// TwinCAT 3 PLC project Struckig_unittest
// ProjectVersion: 0.19.4.0
// ProgramVersion: 3.1.4026.18
// libraries:
//   Struckig, 0.12.2.0 (Stefan Besler)
//   Tc2_System, * (Beckhoff Automation GmbH)
//   Tc3_Module, * (Beckhoff Automation GmbH)
//   TcUnit_Zeugwerk, 1.3.2 (Zeugwerk GmbH)
// project tree:
//   / PlcTask.TcTTO (not stored)
//   POUs/ DebuggedExamplesTest.TcPOU, KnownExamplesSecondOrderTest.TcPOU, MaxVelocitySwitchingTest.TcPOU, Otg1Test.TcPOU, RandomTest.TcPOU, SetVector3.TcPOU (not stored), PropagateTest.TcPOU, VelocityInterfaceTest.TcPOU, MinDurationTest.TcPOU, MathTest.TcPOU, TargetPosTest.TcPOU, TargetPosAccTest.TcPOU, TargetPosVelTest.TcPOU, TargetPosVelAccTest.TcPOU, SecondaryFeaturesTest.TcPOU, CheckCalculation.TcPOU, KnownExamplesTest.TcPOU, MAIN.TcPOU, ZeroLimitsTest.TcPOU
//   Randomizer/ Randomizer.TcPOU (not stored)
//   Random/ IRandom.TcIO (not stored), RandomGaussian.TcPOU, RandomUniform.TcPOU
//   Random/_Test/ RandomGaussianTest.TcPOU (not stored)
// real-time tasks:
//   TASK PlcTask: cycle T#10ms, priority 20, ADS port 350

// ---- POUs/DebuggedExamplesTest.TcPOU
FUNCTION_BLOCK DebuggedExamplesTest EXTENDS TcUnit_Zeugwerk.FB_TestSuite

Test_Trajectory_HasTargetVelocity_HasTargetAcceleration();

METHOD Test_Trajectory_HasTargetVelocity_HasTargetAcceleration
VAR_INST
  ruckig : Struckig.Otg(0.001, 3) := (
  
    Synchronization := SynchronizationType.TimeSync,        
    MaxVelocity := [ 2000.00000000000000000000, 2000.00000000000000000000, 2000.00000000000000000000 ],
    MaxAcceleration := [ 20000.00000000000000000000, 20000.00000000000000000000, 20000.00000000000000000000 ],
    MaxJerk := [ 800000.00000000000000000000, 800000.00000000000000000000, 800000.00000000000000000000 ],
    CurrentPosition := [ -54.94342725690739825950, -71.16344937395382430623, -99.92141940871530891854 ],
    CurrentVelocity := [ 203.04708462957614756306, -87.88615914847480325989, -244.40742200449426491105 ],
    CurrentAcceleration := [ -9414.24830241836389177479, 3433.58972946014000626747, -1048.10905719350193976425 ],
    TargetPosition := [ -30.34627507739200780179, 41.33313071646210801191, 94.47974487226861128875 ],
    TargetVelocity := [ -104.33706621689987059654, -659.36109838358197521302, 811.33117925934993763804 ],
    TargetAcceleration := [ 523.43053514200096287823, 100.75104632855459385610, 320.80199262854853259341 ]
  );
  
  positionExtrema : Struckig.ProfileBound;
END_VAR
TEST('Trajectory_Profile[1]_Step2_TimeVel');

ruckig();

// Check total duration of profiles
AssertEquals_LREAL(Expected := 0.22338925049474450679, Actual := ruckig.Duration, DELTA := 1E-8, Message := 'Duration incorrect');

// Check duration for each phase
positionExtrema := ruckig._profiles[0].Bound();
AssertEquals_LREAL(0.20657109030979783904, positionExtrema.Tmax, 1E-9, message:='Profile[0] Tmax incorrect');
AssertEquals_LREAL(-29.15176131633907630203, positionExtrema.Maximum, 1E-9, message:='Profile[0] maximum incorrect');
AssertEquals_LREAL(0.00000000000000000000, positionExtrema.Tmin, 1E-9, message:='Profile[0] Tmin incorrect');
AssertEquals_LREAL(-54.94342725690739825950, positionExtrema.Minimum, 1E-9, message:='Profile[0] minimum incorrect');

positionExtrema := ruckig._profiles[1].Bound();
AssertEquals_LREAL(0.19826331168683380968, positionExtrema.Tmax, 1E-9, message:='Profile[1] Tmax incorrect');
AssertEquals_LREAL(55.81702313192161568622, positionExtrema.Maximum, 1E-9, message:='Profile[1] maximum incorrect');
AssertEquals_LREAL(0.01113968648909354625, positionExtrema.Tmin, 1E-9, message:='Profile[1] Tmin incorrect');
AssertEquals_LREAL(-71.74511835894615785492, positionExtrema.Minimum, 1E-9, message:='Profile[1] minimum incorrect');

positionExtrema := ruckig._profiles[2].Bound();
AssertEquals_LREAL(0.22338925049474447904, positionExtrema.Tmax, 1E-9, message:='Profile[2] Tmax incorrect');
AssertEquals_LREAL(94.47974487226861128875, positionExtrema.Maximum, 1E-9, message:='Profile[2] maximum incorrect');
AssertEquals_LREAL(0.02606362117094545780, positionExtrema.Tmin, 1E-9, message:='Profile[2] Tmin incorrect');
AssertEquals_LREAL(-104.28684661857214166503, positionExtrema.Minimum, 1E-9, message:='Profile[2] minimum incorrect');
   

TEST_FINISHED();
END_METHOD

END_FUNCTION_BLOCK

// ---- POUs/KnownExamplesSecondOrderTest.TcPOU
FUNCTION_BLOCK KnownExamplesSecondOrderTest EXTENDS TcUnit_Zeugwerk.FB_TestSuite

example01();
example02();
example03();
example04();
example05();
example06();

METHOD example01
VAR_INST
  otg : Struckig.Otg(0.004, 3) := (  
    MaxVelocity :=         [ 1.0, 1.0, 1.0 ],
    MaxAcceleration :=     [ 1.0, 1.0, 1.0 ],
    MaxJerk :=             [ Struckig.Constants.Infinity, Struckig.Constants.Infinity, Struckig.Constants.Infinity ],
    CurrentPosition :=     [ 0.0, -2.0, 0.0 ],
    CurrentVelocity :=     [ 0.0, 0.0, 0.0 ],
    CurrentAcceleration := [ 0.0, 0.0, 0.0 ],
    TargetPosition :=      [ 1.0, -3.0, 2.0 ],
    TargetVelocity :=      [ 0.0, 0.0, 0.0 ],
    TargetAcceleration :=  [ 0.0, 0.0, 0.0 ]
  );
  
END_VAR
TEST('Example-01');

otg();
AssertEquals_LREAL(Expected := 3.0,
             Actual := CheckCalculation(otg),
             DELTA := 1E-8,
             Message := '');
 
TEST_FINISHED();
END_METHOD

METHOD example02
VAR_INST
  otg : Struckig.Otg(0.004, 3) := (  
    MaxVelocity :=         [ 10.0, 10.0, 10.0 ],
    MaxAcceleration :=     [ 1.0, 1.0, 1.0 ],
    CurrentPosition :=     [ 0.0, -2.0, 1.0 ],
    CurrentVelocity :=     [ 0.0, 0.0, 0.0 ],
    CurrentAcceleration := [ 0.0, 0.0, 0.0 ],
    TargetPosition :=      [ 1.0, -3.0, 2.0 ],
    TargetVelocity :=      [ 1.0, 0.0, 0.0 ],
    TargetAcceleration :=  [ 0.0, 0.5, 0.0 ]
  );
  
END_VAR
TEST('Example-02');

otg();
AssertEquals_LREAL(Expected := 2.0,
             Actual := CheckCalculation(otg),
             Delta := 1E-8,
             Message := '');
 
TEST_FINISHED();
END_METHOD

METHOD example03
VAR_INST
  otg : Struckig.Otg(0.004, 3) := (  
    MaxVelocity :=         [ 10.0, 10.0, 10.0 ],
    MaxAcceleration :=     [ 1.0, 1.0, 1.0 ],
    CurrentPosition :=     [ 0.0, -2.0, -2.0 ],
    CurrentVelocity :=     [ 0.1, 0.1, 1.0 ],
    CurrentAcceleration := [ 0.0, 0.0, 0.0 ],
    TargetPosition :=      [ 1.0, -3.0, 2.0 ],
    TargetVelocity :=      [ 1.0, 0.0, 0.0 ],
    TargetAcceleration :=  [ 0.0, 0.5, 0.0 ]
  );
  
END_VAR
TEST('Example-03');

otg();
AssertEquals_LREAL(Expected := 3.24264068711928,
             Actual := CheckCalculation(otg),
             DELTA := 1E-8,
             Message := '');
 
TEST_FINISHED();
END_METHOD

METHOD example04
VAR_INST
  otg : Struckig.Otg(0.004, 3) := (       
    MaxVelocity :=         [ 10.0, 10.0, 10.0 ],
    MaxAcceleration :=     [ 1.0, 1.0, 1.0 ],
    CurrentPosition :=     [ 0.0, 0.0, 0.0 ],
    CurrentVelocity :=     [ 0.0, 1.0, 0.0 ],
    CurrentAcceleration := [ 0.0, 0.0, 0.0 ],
    TargetPosition :=      [ 0.0, 0.0, 0.0 ],
    TargetVelocity :=      [ 0.0, 1.0, 0.0 ],
    TargetAcceleration :=  [ 0.0, 0.0, 0.0 ]
  );
  
  
END_VAR
TEST('Example-04');

otg();
AssertEquals_LREAL(Expected := 0.0,
             Actual := CheckCalculation(otg),
             DELTA := 1E-8,
             Message := '');
 
TEST_FINISHED();
END_METHOD

METHOD example05
VAR_INST
  otg : Struckig.Otg(0.004, 3) := (  
    MaxVelocity :=         [ 10.0, 10.0, 10.0 ],
    MaxAcceleration :=     [ 1.0, 1.0, 1.0 ],
    CurrentPosition :=     [ 0.0, 0.0, 0.0 ],
    CurrentVelocity :=     [ 0.0, 1.0, 0.0 ],
    CurrentAcceleration := [ 0.0, 0.0, 0.0 ],
    TargetPosition :=      [ 0.0, 1E-4, 0.0 ],
    TargetVelocity :=      [ 0.0, 1.0, 0.0 ],
    TargetAcceleration :=  [ 0.0, 0.0, 0.0 ]
  );
  
END_VAR
TEST('Example-05');

otg();
AssertEquals_LREAL(Expected := 0.0001,
             Actual := CheckCalculation(otg),
             DELTA := 1E-8,
             Message := '');
 
TEST_FINISHED();
END_METHOD

METHOD example06
VAR_INST
  otg : Struckig.Otg(0.004, 3) := (  
    MaxVelocity :=         [ 10.0, 10.0, 10.0 ],
    MaxAcceleration :=     [ 1.0, 1.0, 1.0 ],
    CurrentPosition :=     [ 0.0, 0.0, 0.0 ],
    CurrentVelocity :=     [ 0.0, 1.0, 0.0 ],
    CurrentAcceleration := [ 0.0, 0.0, 0.0 ],
    TargetPosition :=      [ 1E-4, 0.0, 0.0 ],
    TargetVelocity :=      [ 0.0, 1.0, 0.0 ],
    TargetAcceleration :=  [ 0.0, 0.0, 0.0 ]
  );
  
END_VAR
TEST('Example-06');

otg();
AssertEquals_LREAL(Expected := 4.0,
             Actual := CheckCalculation(otg),
             DELTA := 1E-8,
             Message := '');
 
TEST_FINISHED();
END_METHOD

END_FUNCTION_BLOCK

// ---- POUs/CheckCalculation.TcPOU
FUNCTION CheckCalculation : LREAL
VAR_INPUT
  otg : Struckig.IOtg;
END_VAR

REPEAT 
  otg.Cyclic();
  otg.PassOutputToInput();
UNTIL otg.State <> Struckig.TrajectoryState.Busy END_REPEAT

CheckCalculation := otg.Duration;

END_FUNCTION

// ---- POUs/MaxVelocitySwitchingTest.TcPOU
FUNCTION_BLOCK MaxVelocitySwitchingTest EXTENDS TcUnit_Zeugwerk.FB_TestSuite

Test_Trajectory();
Test_SmoothBrake_DuringAccel();
Test_SmoothBrake_FromCruise();
Test_SmoothBrake_Disabled();
Test_SmoothBrake_ReachesNewVelocity();

METHOD Test_SmoothBrake_Disabled
VAR_INST
  otg : Struckig.Otg(0.001, 1) := (
    Synchronization := SynchronizationType.TimeSync,
    SmoothBrake := FALSE,
    MaxVelocity := [ 1000 ],
    MaxAcceleration := [ 5000 ],
    MaxJerk := [ 50000 ],
    CurrentPosition := [ 0 ],
    CurrentVelocity := [ 0 ],
    CurrentAcceleration := [ 0 ],
    TargetPosition := [ 50000 ],
    TargetVelocity := [ 0 ],
    TargetAcceleration := [ 0 ]
  );
END_VAR
TEST('SmoothBrake_Disabled');

otg();

REPEAT 
  otg.Cyclic();
  otg.PassOutputToInput();
UNTIL otg.CurrentTime >= otg._profiles[0].t_sum[2] + 0.05 END_REPEAT

otg.MaxVelocity[0] := 500;

REPEAT 
  otg.Cyclic();
  otg.PassOutputToInput();
UNTIL otg.State <> Struckig.TrajectoryState.Busy END_REPEAT

AssertTrue(otg.State <> Struckig.TrajectoryState.Error, Message := 'Legacy mode (SmoothBrake=FALSE) must complete without error');

TEST_FINISHED();
END_METHOD

METHOD Test_SmoothBrake_DuringAccel
VAR_INST
  otg : Struckig.Otg(0.001, 1) := (
    Synchronization := SynchronizationType.TimeSync,
    SmoothBrake := TRUE,
    MaxVelocity := [ 1000 ],
    MaxAcceleration := [ 5000 ],
    MaxJerk := [ 50000 ],
    CurrentPosition := [ 0 ],
    CurrentVelocity := [ 0 ],
    CurrentAcceleration := [ 0 ],
    TargetPosition := [ 50000 ],
    TargetVelocity := [ 0 ],
    TargetAcceleration := [ 0 ]
  );
END_VAR
VAR_INST
  minV : LREAL;
END_VAR
TEST('SmoothBrake_DuringAccel');

otg();

REPEAT 
  otg.Cyclic();
  otg.PassOutputToInput();
UNTIL otg.NewVelocity[0] > 900 OR_ELSE otg.CurrentTime > 5.0 END_REPEAT

otg.MaxVelocity[0] := 500;

minV := 1000;
REPEAT 
  otg.Cyclic();
  IF otg.CurrentTime < otg._profiles[0].Brake.Duration + otg._profiles[0].t_sum[3] THEN
    IF otg.NewVelocity[0] < minV THEN
      minV := otg.NewVelocity[0];
    END_IF
  END_IF
  otg.PassOutputToInput();
UNTIL otg.State <> Struckig.TrajectoryState.Busy END_REPEAT

AssertTrue(otg.State <> Struckig.TrajectoryState.Error, Message := 'OTG must not enter Error state');
AssertTrue(minV > 400.0, Message := 'During accel, velocity must not dip far below new MaxVelocity (500)');

TEST_FINISHED();
END_METHOD

METHOD Test_SmoothBrake_FromCruise
VAR_INST
  otg : Struckig.Otg(0.001, 1) := (
    Synchronization := SynchronizationType.TimeSync,
    SmoothBrake := TRUE,
    MaxVelocity := [ 1000 ],
    MaxAcceleration := [ 5000 ],
    MaxJerk := [ 50000 ],
    CurrentPosition := [ 0 ],
    CurrentVelocity := [ 0 ],
    CurrentAcceleration := [ 0 ],
    TargetPosition := [ 50000 ],
    TargetVelocity := [ 0 ],
    TargetAcceleration := [ 0 ]
  );
END_VAR
VAR
  minV : LREAL;
END_VAR
TEST('SmoothBrake_FromCruise');

otg();

REPEAT 
  otg.Cyclic();
  otg.PassOutputToInput();
UNTIL otg.CurrentTime >= otg._profiles[0].t_sum[2] + 0.05 END_REPEAT

otg.MaxVelocity[0] := 500;

minV := 1000;
REPEAT 
  otg.Cyclic();
  IF otg.CurrentTime < otg._profiles[0].Brake.Duration + otg._profiles[0].t_sum[3] THEN
    IF otg.NewVelocity[0] < minV THEN
      minV := otg.NewVelocity[0];
    END_IF
  END_IF
  otg.PassOutputToInput();
UNTIL otg.State <> Struckig.TrajectoryState.Busy END_REPEAT

AssertTrue(otg.State <> Struckig.TrajectoryState.Error, Message := 'OTG must not enter Error state');
AssertTrue(minV > 400.0, Message := 'From cruise, velocity must not dip far below new MaxVelocity (500)');

TEST_FINISHED();
END_METHOD

METHOD Test_SmoothBrake_ReachesNewVelocity
VAR_INST
  otg : Struckig.Otg(0.001, 1) := (
    Synchronization := SynchronizationType.TimeSync,
    SmoothBrake := TRUE,
    MaxVelocity := [ 1000 ],
    MaxAcceleration := [ 5000 ],
    MaxJerk := [ 50000 ],
    CurrentPosition := [ 0 ],
    CurrentVelocity := [ 0 ],
    CurrentAcceleration := [ 0 ],
    TargetPosition := [ 50000 ],
    TargetVelocity := [ 0 ],
    TargetAcceleration := [ 0 ]
  );
END_VAR
VAR
  vAfter : LREAL;
  captured : BOOL;
END_VAR
TEST('SmoothBrake_ReachesNewVelocity');

otg();

REPEAT 
  otg.Cyclic();
  otg.PassOutputToInput();
UNTIL otg.CurrentTime >= otg._profiles[0].t_sum[2] + 0.05 END_REPEAT

otg.MaxVelocity[0] := 500;

captured := FALSE;
REPEAT 
  otg.Cyclic();
  IF NOT captured AND_THEN otg.CurrentTime >= otg._profiles[0].Brake.Duration + otg._profiles[0].t_sum[2] + 0.01 THEN
    vAfter := otg.NewVelocity[0];
    captured := TRUE;
  END_IF
  otg.PassOutputToInput();
UNTIL otg.State <> Struckig.TrajectoryState.Busy END_REPEAT

AssertTrue(otg.State <> Struckig.TrajectoryState.Error, Message := 'OTG must not enter Error state');
AssertTrue(vAfter > 490.0 AND_THEN vAfter < 510.0, Message := 'After transition, velocity should settle at new MaxVelocity (~500)');

TEST_FINISHED();
END_METHOD

METHOD Test_Trajectory
VAR_INST
  ruckig : Struckig.Otg(0.001, 1) := (
    Synchronization := SynchronizationType.TimeSync,        
    MaxVelocity := [ 10000.00000000000000000000 ],
    MaxAcceleration := [ 20000.00000000000000000000 ],
    MaxJerk := [ 800000.00000000000000000000 ],
    CurrentPosition := [ 0 ],
    CurrentVelocity := [ 0 ],
    CurrentAcceleration := [ 0 ],
    TargetPosition := [ 10000 ],
    TargetVelocity := [ 0 ],
    TargetAcceleration := [ 0 ]
  );
  
END_VAR
TEST('Trajectory');

ruckig();

REPEAT 
  ruckig.Cyclic();
  ruckig.PassOutputToInput();
UNTIL ruckig.CurrentTime >= ruckig._profiles[0].t_sum[2] + 0.05 END_REPEAT

ruckig.MaxVelocity[0] := 9500;

REPEAT 
  ruckig.Cyclic();
  ruckig.PassOutputToInput();
UNTIL ruckig.State <> Struckig.TrajectoryState.Busy END_REPEAT

TEST_FINISHED();
END_METHOD

END_FUNCTION_BLOCK

// ---- POUs/Otg1Test.TcPOU
FUNCTION_BLOCK Otg1Test EXTENDS TcUnit_Zeugwerk.FB_TestSuite

example06();

METHOD example06
VAR_INST
  otg1 : Struckig.Otg1(0.005) := (
  
    Synchronization := SynchronizationType.None,        
    MaxVelocity :=          0.4,
    MaxAcceleration :=      1.0,
    MaxJerk :=              2.0,
    CurrentPosition :=      0.0,
    CurrentVelocity :=      0.0,
    CurrentAcceleration :=  0.0,
    TargetPosition :=       1.0,
    TargetVelocity :=       0.0,
    TargetAcceleration :=   0.0
  );
  	
END_VAR
TEST('Example-06');

otg1();
AssertEquals_LREAL(Expected := 3.394427191,
             Actual := CheckCalculation(otg1),
             DELTA := 1E-8,
             Message := '');
 
TEST_FINISHED();
END_METHOD

END_FUNCTION_BLOCK

// ---- POUs/RandomTest.TcPOU
FUNCTION_BLOCK RandomTest EXTENDS TcUnit_Zeugwerk.FB_TestSuite
VAR
  _number_trajectories : UDINT := 256 * 1024; // Some user variable you want to be able to set
  _position_random_3 : UDINT  := MIN(250000, _number_trajectories / 25);  
  _velocity_random_3 : UDINT  := MIN(250000, _number_trajectories / 25);
  
  _positionDist : RandomGaussian(seed:=45, mu:=0, sigma:=4);
  _dynamicDist : RandomGaussian(seed:=46, mu:=0, sigma:=0.8);
  _limitDist : RandomUniform(seed:=47, lowerBound:=0.08, upperBound:=16.0);
  _limitDistHigh : RandomUniform(seed:=48, lowerBound:=10, upperBound:=1000000.0);
  _minLimitDist : RandomUniform(seed:=49, lowerBound:=-16, upperBound:=-0.08);

END_VAR

Test_PositionFirstRandom3();

Test_VelocitySecondRandom3();
Test_PositionSecondRandom3();

Test_VelocityThirdRandom3();
Test_PositionThirdRandom3();

METHOD Test_PositionFirstRandom3
VAR_INST
  p : Randomizer(_positionDist);
  d : Randomizer(_dynamicDist);
  l : Randomizer(_limitDist);
  
  otg : Struckig.Otg(0.005, 3) := (
    ControlInterface := ControlInterfaceType.Position
  );
   
END_VAR
VAR
  i : UDINT;
END_VAR
TEST('Test_PositionFirstRandom3');

FOR i:=0 TO _position_random_3
DO

  IF i < _position_random_3 / 2
  THEN
    otg.Synchronization := SynchronizationType.Phase;
  ELSE
    otg.Synchronization := SynchronizationType.TimeSync;    
  END_IF
  
  IF i < _position_random_3 / 20
  THEN
    otg.Discretization := DiscretizationType.Discrete;
  ELSE
    otg.Discretization := DiscretizationType.Continuous;    
  END_IF  

  p.Fill(ADR(otg.CurrentPosition), 3);
  d.FillOrZero(ADR(otg.CurrentVelocity), 3, 0.9);
  d.FillOrZero(ADR(otg.CurrentAcceleration), 3, 0.9);
  
  p.Fill(ADR(otg.TargetPosition), 3);
  d.FillOrZero(ADR(otg.TargetVelocity), 3, 0.7);
  d.FillOrZero(ADR(otg.TargetAcceleration), 3, 0.6);
  
  l.FillMax(ADR(otg.MaxVelocity), 3, ADR(otg.TargetVelocity));
  
  IF NOT otg.ValidateInput(FALSE, TRUE)
  THEN
    i := i - 1;
  END_IF
  
  CheckCalculation(otg);
  
END_FOR

TEST_FINISHED();
END_METHOD

METHOD Test_PositionSecondRandom3
VAR_INST
  p : Randomizer(_positionDist);
  d : Randomizer(_dynamicDist);
  l : Randomizer(_limitDist);
  

  otg : Struckig.Otg(0.005, 3) := (
    ControlInterface := ControlInterfaceType.Position
  );
   
END_VAR
VAR
  i : UDINT;
END_VAR
TEST('Test_PositionSecondRandom3');

FOR i:=0 TO _position_random_3
DO

  IF i < _position_random_3 / 2
  THEN
    otg.Synchronization := SynchronizationType.Phase;
  ELSE
    otg.Synchronization := SynchronizationType.TimeSync;    
  END_IF
  
  IF i < _position_random_3 / 20
  THEN
    otg.Discretization := DiscretizationType.Discrete;
  ELSE
    otg.Discretization := DiscretizationType.Continuous;    
  END_IF  

  p.Fill(ADR(otg.CurrentPosition), 3);
  d.FillOrZero(ADR(otg.CurrentVelocity), 3, 0.9);
  d.FillOrZero(ADR(otg.CurrentAcceleration), 3, 0.9);
  
  p.Fill(ADR(otg.TargetPosition), 3);
  d.FillOrZero(ADR(otg.TargetVelocity), 3, 0.7);
  d.FillOrZero(ADR(otg.TargetAcceleration), 3, 0.6);
  
  l.FillMax(ADR(otg.MaxVelocity), 3, ADR(otg.TargetVelocity));
  l.FillMax(ADR(otg.MaxAcceleration), 3, ADR(otg.TargetAcceleration));
  
  IF NOT otg.ValidateInput(FALSE, TRUE)
  THEN
    i := i - 1;
  END_IF
  
  CheckCalculation(otg);
  
END_FOR

TEST_FINISHED();
END_METHOD

METHOD Test_PositionThirdRandom3
VAR_INST
  p : Randomizer(_positionDist);
  d : Randomizer(_dynamicDist);
  l : Randomizer(_limitDist);
  

  otg : Struckig.Otg(0.005, 3) := (
    ControlInterface := ControlInterfaceType.Position
  );
   
END_VAR
VAR
  i : UDINT;
END_VAR
TEST('Test_PositionThirdRandom3');

FOR i:=0 TO _position_random_3
DO

  IF i < _position_random_3 / 2
  THEN
    otg.Synchronization := SynchronizationType.Phase;
  ELSE
    otg.Synchronization := SynchronizationType.TimeSync;    
  END_IF
  
  IF i < _position_random_3 / 20
  THEN
    otg.Discretization := DiscretizationType.Discrete;
  ELSE
    otg.Discretization := DiscretizationType.Continuous;    
  END_IF  

  p.Fill(ADR(otg.CurrentPosition), 3);
  d.FillOrZero(ADR(otg.CurrentVelocity), 3, 0.9);
  d.FillOrZero(ADR(otg.CurrentAcceleration), 3, 0.9);
  
  p.Fill(ADR(otg.TargetPosition), 3);
  d.FillOrZero(ADR(otg.TargetVelocity), 3, 0.7);
  d.FillOrZero(ADR(otg.TargetAcceleration), 3, 0.6);
  
  l.FillMax(ADR(otg.MaxVelocity), 3, ADR(otg.TargetVelocity));
  l.FillMax(ADR(otg.MaxAcceleration), 3, ADR(otg.TargetAcceleration));
  l.Fill(ADR(otg.MaxJerk), 3);  
  
  IF NOT otg.ValidateInput(FALSE, TRUE)
  THEN
    i := i - 1;
  END_IF
  
  CheckCalculation(otg);
  
END_FOR

TEST_FINISHED();
END_METHOD

METHOD Test_VelocitySecondRandom3
VAR_INST
  p : Randomizer(_positionDist);
  d : Randomizer(_dynamicDist);
  l : Randomizer(_limitDist);
  min_l : Randomizer(_minLimitDist);
  

  otg : Struckig.Otg(0.005, 3) := (
    ControlInterface := ControlInterfaceType.Velocity
  );
   
END_VAR
VAR
  i : UDINT;
END_VAR
TEST('Test_VelocitySecondRandom3');

otg.CurrentPosition[0] := 0;
otg.CurrentPosition[1] := 0;
otg.CurrentPosition[2] := 0;

FOR i:=0 TO _velocity_random_3
DO
  d.FillOrZero(ADR(otg.CurrentVelocity), 3, 0.9);
  d.FillOrZero(ADR(otg.CurrentAcceleration), 3, 0.9);
  d.FillOrZero(ADR(otg.TargetVelocity), 3, 0.9);
  d.FillOrZero(ADR(otg.TargetAcceleration), 3, 0.9);
  l.FillMax(ADR(otg.MaxAcceleration), 3, ADR(otg.TargetAcceleration));
  
  CheckCalculation(otg);
  
END_FOR

TEST_FINISHED();
END_METHOD

METHOD Test_VelocityThirdRandom3
VAR_INST
  p : Randomizer(_positionDist);
  d : Randomizer(_dynamicDist);
  l : Randomizer(_limitDist);
  min_l : Randomizer(_minLimitDist);
  

  otg : Struckig.Otg(0.005, 3) := (
    ControlInterface := ControlInterfaceType.Velocity
  );
   
END_VAR
VAR
  i : UDINT;
END_VAR
TEST('Test_VelocityThirddRandom3');

otg.CurrentPosition[0] := 0;
otg.CurrentPosition[1] := 0;
otg.CurrentPosition[2] := 0;

FOR i:=0 TO _velocity_random_3
DO
  d.FillOrZero(ADR(otg.CurrentVelocity), 3, 0.9);
  d.FillOrZero(ADR(otg.CurrentAcceleration), 3, 0.9);
  d.FillOrZero(ADR(otg.TargetVelocity), 3, 0.9);
  d.FillOrZero(ADR(otg.TargetAcceleration), 3, 0.9);
  l.FillMax(ADR(otg.MaxAcceleration), 3, ADR(otg.TargetAcceleration));
  l.Fill(ADR(otg.MaxJerk), 3);
  
  CheckCalculation(otg);
  
END_FOR

TEST_FINISHED();
END_METHOD

END_FUNCTION_BLOCK

// ---- Random/RandomGaussian.TcPOU
FUNCTION_BLOCK RandomGaussian IMPLEMENTS IRandom
VAR
  _mu : LREAL;
  _sigma : LREAL;    
  _rnd : Tc2_System.DRAND;
END_VAR

METHOD FB_init : BOOL
VAR_INPUT
	bInitRetains : BOOL; // if TRUE, the retain variables are initialized (warm start / cold start)
	bInCopyCode : BOOL;  // if TRUE, the instance afterwards gets moved into the copy code (online change)
  seed : INT;  
  mu : LREAL;
  sigma : LREAL;
END_VAR
SetSeed(seed);
SetMean(mu);
SetSigma(sigma);
END_METHOD

/// Implementation of the Box-Muller transform for normal distributed random
/// variables. There are much faster methods for doing this.
/// Implementation taken from [here](https://en.wikipedia.org/wiki/Box%E2%80%93Muller_transform)
METHOD Next : LREAL
VAR
  u1, u2 : LREAL;
END_VAR
VAR CONSTANT
  Pi : LREAL := 3.14159265358979323846;
END_VAR
//create two random numbers, make sure u1 is greater than epsilon
REPEAT
  _rnd(Num => u1);
  _rnd(Num => u2);  
UNTIL u1 > 1E-8 END_REPEAT

//compute z0 and z1
Next  := (_sigma * SQRT(-2.0 * LOG(u1))) * COS(2*Pi * u2) + _mu;

// we do not need the 2nd randomly distributed variable
// z1 := mag * SIN(2*Struckig.Constants.Pi  * u2) + mu;
END_METHOD

METHOD FINAL SetMean
VAR_INPUT
  mu : LREAL;
END_VAR
_mu := mu;
END_METHOD

METHOD FINAL SetSeed
VAR_INPUT
  seed : INT;
END_VAR
_rnd.Seed := seed;
END_METHOD

METHOD FINAL SetSigma
VAR_INPUT
  sigma : LREAL;
END_VAR
_sigma := sigma;
END_METHOD

END_FUNCTION_BLOCK

// ---- Random/RandomUniform.TcPOU
FUNCTION_BLOCK RandomUniform IMPLEMENTS IRandom
VAR
  _lowerBound : LREAL;
  _upperBound : LREAL;  
  _rnd : Tc2_System.DRAND;
END_VAR

METHOD FB_init : BOOL
VAR_INPUT
	bInitRetains : BOOL; // if TRUE, the retain variables are initialized (warm start / cold start)
	bInCopyCode : BOOL;  // if TRUE, the instance afterwards gets moved into the copy code (online change)
  seed : INT;      
  lowerBound : LREAL;
  upperBound : LREAL;
END_VAR
SetSeed(seed);
SetBounds(lowerBound, upperBound);
END_METHOD

METHOD Next : LREAL
_rnd();
Next := _rnd.Num * (_upperBound-_lowerBound) + _lowerBound;
END_METHOD

METHOD FINAL SetBounds
VAR_INPUT
  lowerBound : LREAL;
  upperBound : LREAL;
END_VAR
_lowerBound := lowerBound;
_upperBound := upperBound;
END_METHOD

METHOD FINAL SetSeed
VAR_INPUT
  seed : INT;
END_VAR
_rnd.Seed := seed;
END_METHOD

END_FUNCTION_BLOCK

// ---- POUs/PropagateTest.TcPOU
FUNCTION_BLOCK PropagateTest EXTENDS TcUnit_Zeugwerk.FB_TestSuite

Test_AutoPropagate();
Test_ManualPropagate();
Test_NoPropagate();

METHOD Test_AutoPropagate
VAR_INST
  ruckig : Struckig.Otg(0.001, 3) := (
  
    Synchronization := SynchronizationType.TimeSync,        
    MaxVelocity := [ 2000, 2000, 2000 ],
    MaxAcceleration := [ 20000, 20000, 20000 ],
    MaxJerk := [ 8000, 80000, 800000 ],
    CurrentPosition := [ 0,0,0  ],
    CurrentVelocity := [ 0,0,0 ],
    CurrentAcceleration := [ 0,0,0 ],
    TargetPosition := [ 1, 10, 100 ],
    TargetVelocity := [ 0,0,0 ],
    TargetAcceleration := [ 0,0,0 ]
  );
  
  StartPosition, StartVelocity, StartAcceleration : ARRAY[0..ParameterList.MaxDoFs] OF LREAL; // Current state
  NewPosition, NewVelocity, NewAcceleration : ARRAY[0..ParameterList.MaxDoFs] OF LREAL; // Current state  
END_VAR
TEST('Test_AutoPropagate');

StartPosition := ruckig.CurrentPosition;
StartVelocity := ruckig.CurrentVelocity;
StartAcceleration := ruckig.CurrentAcceleration;

ruckig();
AssertTrue(0 = ruckig.CurrentPosition[0], Message:=''); 

NewPosition := ruckig.NewPosition;
NewVelocity := ruckig.NewVelocity;
NewAcceleration := ruckig.NewAcceleration;

ruckig(EnableAutoPropagate := TRUE);

AssertTrue(0 <> ruckig.CurrentPosition[0], Message:=''); 
AssertArrayEquals_LREAL(Expecteds:=NewPosition, Actuals:=ruckig.CurrentPosition, Delta:=1E-6, Message:='');
AssertArrayEquals_LREAL(Expecteds:=NewVelocity, Actuals:=ruckig.CurrentVelocity, Delta:=1E-6, Message:='');
AssertArrayEquals_LREAL(Expecteds:=NewAcceleration, Actuals:=ruckig.CurrentAcceleration, Delta:=1E-6, Message:='');

TEST_FINISHED();
END_METHOD

METHOD Test_ManualPropagate
VAR_INST
  ruckig : Struckig.Otg(0.001, 3) := (
  
    Synchronization := SynchronizationType.TimeSync,        
    MaxVelocity := [ 2000, 2000, 2000 ],
    MaxAcceleration := [ 20000, 20000, 20000 ],
    MaxJerk := [ 8000, 80000, 800000 ],
    CurrentPosition := [ 0,0,0  ],
    CurrentVelocity := [ 0,0,0 ],
    CurrentAcceleration := [ 0,0,0 ],
    TargetPosition := [ 1, 10, 100 ],
    TargetVelocity := [ 0,0,0 ],
    TargetAcceleration := [ 0,0,0 ]
  );
  
  StartPosition, StartVelocity, StartAcceleration : ARRAY[0..ParameterList.MaxDoFs] OF LREAL; // Current state
  NewPosition, NewVelocity, NewAcceleration : ARRAY[0..ParameterList.MaxDoFs] OF LREAL; // Current state  
END_VAR
TEST('Test_ManualPropagate');

StartPosition := ruckig.CurrentPosition;
StartVelocity := ruckig.CurrentVelocity;
StartAcceleration := ruckig.CurrentAcceleration;

ruckig();
AssertTrue(0 = ruckig.CurrentPosition[0], Message:=''); 

NewPosition := ruckig.NewPosition;
NewVelocity := ruckig.NewVelocity;
NewAcceleration := ruckig.NewAcceleration;

ruckig.PassOutputToInput();

AssertTrue(0 <> ruckig.CurrentPosition[0], Message:=''); 
AssertArrayEquals_LREAL(Expecteds:=NewPosition, Actuals:=ruckig.CurrentPosition, Delta:=1E-6, Message:='');
AssertArrayEquals_LREAL(Expecteds:=NewVelocity, Actuals:=ruckig.CurrentVelocity, Delta:=1E-6, Message:='');
AssertArrayEquals_LREAL(Expecteds:=NewAcceleration, Actuals:=ruckig.CurrentAcceleration, Delta:=1E-6, Message:='');

TEST_FINISHED();
END_METHOD

METHOD Test_NoPropagate
VAR_INST
  ruckig : Struckig.Otg(0.001, 3) := (
  
    Synchronization := SynchronizationType.TimeSync,        
    MaxVelocity := [ 2000, 2000, 2000 ],
    MaxAcceleration := [ 20000, 20000, 20000 ],
    MaxJerk := [ 8000, 80000, 800000 ],
    CurrentPosition := [ 0,0,0  ],
    CurrentVelocity := [ 0,0,0 ],
    CurrentAcceleration := [ 0,0,0 ],
    TargetPosition := [ 1, 10, 100 ],
    TargetVelocity := [ 0,0,0 ],
    TargetAcceleration := [ 0,0,0 ]
  );
  
  StartPosition, StartVelocity, StartAcceleration : ARRAY[0..ParameterList.MaxDoFs] OF LREAL; // Current state
  NewPosition, NewVelocity, NewAcceleration : ARRAY[0..ParameterList.MaxDoFs] OF LREAL; // Current state  
END_VAR
TEST('Test_NoPropagate');

StartPosition := ruckig.CurrentPosition;
StartVelocity := ruckig.CurrentVelocity;
StartAcceleration := ruckig.CurrentAcceleration;

AssertArrayEquals_LREAL(Expecteds:=StartPosition, Actuals:=ruckig.CurrentPosition, Delta:=1E-6, Message:='');
AssertArrayEquals_LREAL(Expecteds:=StartVelocity, Actuals:=ruckig.CurrentVelocity, Delta:=1E-6, Message:='');
AssertArrayEquals_LREAL(Expecteds:=StartAcceleration, Actuals:=ruckig.CurrentAcceleration, Delta:=1E-6, Message:='');

ruckig();

AssertArrayEquals_LREAL(Expecteds:=StartPosition, Actuals:=ruckig.CurrentPosition, Delta:=1E-6, Message:='');
AssertArrayEquals_LREAL(Expecteds:=StartVelocity, Actuals:=ruckig.CurrentVelocity, Delta:=1E-6, Message:='');
AssertArrayEquals_LREAL(Expecteds:=StartAcceleration, Actuals:=ruckig.CurrentAcceleration, Delta:=1E-6, Message:='');

TEST_FINISHED();
END_METHOD

END_FUNCTION_BLOCK

// ---- POUs/VelocityInterfaceTest.TcPOU
FUNCTION_BLOCK VelocityInterfaceTest EXTENDS TcUnit_Zeugwerk.FB_TestSuite
VAR
  ruckig : Struckig.Otg(0.001, 3) := (
  
    ControlInterface := ControlInterfaceType.Velocity,
    Synchronization := SynchronizationType.TimeSync,
    MinDuration := 1.0,
    MaxVelocity := [ 2000.0, 2000.0, 2000.0 ],
    MaxAcceleration := [ 20000.0, 20000.0, 20000.0 ],
    MaxJerk := [ 800000.0, 800000.0, 800000.0 ],
    CurrentPosition := [ 84.42864058696819, -11.7964257097819, -59.92935947897627 ],
    CurrentVelocity := [ 270.39639434509445, -161.39803590006613, -753.5522105491483 ],
    CurrentAcceleration := [ -4592.668311850281, 5244.516031969961, 5496.025200940228 ],
    TargetPosition := [ 10.638869224719016, -12.72927242305046, -23.99107805858567 ],
    TargetVelocity := [ 0.0, 0.0, 0.0 ],
    TargetAcceleration := [ 0.0, 0.0, 0.0 ]
  );
  
  positionExtrema : Struckig.ProfileBound;	
END_VAR

Test_Trajectory_VelIntrf_HasMinDuration_HasTargetVelocity_HasTargetAcceleration_1();
Test_Trajectory_VelIntrf_HasMinDuration_HasTargetAcceleration_2();
Test_Trajectory_VelIntrf_HasMinDuration_3();
Test_Trajectory_VelIntrf_HasMinDuration_4();
Test_Trajectory_VelIntrf_HasMinDuration_HasTargetVelocity_5();
Test_Trajectory_VelIntrf_HasMinDuration_6();
Test_Trajectory_VelIntrf_HasMinDuration_HasTargetVelocity_7();
Test_Trajectory_VelIntrf_HasMinDuration_8();
Test_Trajectory_VelIntrf_HasMinDuration_HasTargetVelocity_HasTargetAcceleration_9();
Test_Trajectory_VelIntrf_HasMinDuration_HasTargetVelocity_10();
Test_Trajectory_VelIntrf_HasMinDuration_11();
Test_Trajectory_VelIntrf_HasMinDuration_HasTargetAcceleration_12();
Test_Trajectory_VelIntrf_HasMinDuration_13();
Test_Trajectory_VelIntrf_HasMinDuration_HasTargetAcceleration_14();
Test_Trajectory_VelIntrf_HasMinDuration_HasTargetAcceleration_15();
Test_Trajectory_VelIntrf_HasMinDuration_16();
Test_Trajectory_VelIntrf_HasMinDuration_HasTargetVelocity_HasTargetAcceleration_17();
Test_Trajectory_VelIntrf_HasMinDuration_18();
Test_Trajectory_VelIntrf_HasMinDuration_HasTargetVelocity_HasTargetAcceleration_19();
Test_Trajectory_VelIntrf_HasMinDuration_HasTargetVelocity_HasTargetAcceleration_20();
Test_Trajectory_VelIntrf_HasMinDuration_HasTargetVelocity_HasTargetAcceleration_21();
Test_Trajectory_VelIntrf_HasMinDuration_HasTargetVelocity_HasTargetAcceleration_22();
Test_Trajectory_VelIntrf_HasMinDuration_HasTargetVelocity_HasTargetAcceleration_23();
Test_Trajectory_VelIntrf_HasMinDuration_HasTargetAcceleration_24();
Test_Trajectory_VelIntrf_HasMinDuration_HasTargetVelocity_HasTargetAcceleration_25();
Test_Trajectory_VelIntrf_HasMinDuration_HasTargetVelocity_HasTargetAcceleration_26();
Test_Trajectory_VelIntrf_HasMinDuration_27();
Test_Trajectory_VelIntrf_HasMinDuration_HasTargetAcceleration_28();
Test_Trajectory_VelIntrf_HasMinDuration_HasTargetVelocity_29();
Test_Trajectory_VelIntrf_HasMinDuration_30();
Test_Trajectory_VelIntrf_HasMinDuration_HasTargetVelocity_31();
Test_Trajectory_VelIntrf_HasMinDuration_32();
Test_Trajectory_VelIntrf_HasMinDuration_HasTargetVelocity_HasTargetAcceleration_33();
Test_Trajectory_VelIntrf_HasMinDuration_34();
Test_Trajectory_VelIntrf_HasMinDuration_HasTargetVelocity_35();
Test_Trajectory_VelIntrf_HasMinDuration_36();
Test_Trajectory_VelIntrf_HasMinDuration_HasTargetVelocity_HasTargetAcceleration_37();
Test_Trajectory_VelIntrf_HasMinDuration_38();
Test_Trajectory_VelIntrf_HasMinDuration_39();
Test_Trajectory_VelIntrf_HasMinDuration_HasTargetVelocity_HasTargetAcceleration_40();

METHOD Test_Trajectory_VelIntrf_HasMinDuration_11
VAR_INST
  ruckig : Struckig.Otg(0.001, 3) := (
  
    ControlInterface := ControlInterfaceType.Velocity,
    Synchronization := SynchronizationType.TimeSync,
    MinDuration := 2.0,
    MaxVelocity := [ 2000.0, 2000.0, 2000.0 ],
    MaxAcceleration := [ 20000.0, 20000.0, 20000.0 ],
    MaxJerk := [ 800000.0, 800000.0, 800000.0 ],
    CurrentPosition := [ 77.60057317918495, 30.762778737727984, 64.62813070858635 ],
    CurrentVelocity := [ 277.63976330079527, 532.4341040614261, 390.8302995848069 ],
    CurrentAcceleration := [ 9592.953817598162, 637.6679138078889, 9538.484770013067 ],
    TargetPosition := [ 26.576937052679654, 55.39866329991938, -59.04906710553117 ],
    TargetVelocity := [ 0.0, 0.0, 0.0 ],
    TargetAcceleration := [ 0.0, 0.0, 0.0 ]
  );
  
  positionExtrema : Struckig.ProfileBound;
END_VAR
TEST('Trajectory_VelIntrf_HasMinDuration_11');

ruckig();

// Check total duration of profiles
AssertEquals_LREAL(Expected := 2.0, Actual := ruckig.Duration, DELTA := 1E-8, Message := 'Duration incorrect');

// Check minimum duration
AssertEquals_LREAL(Expected := ruckig.MinDuration, Actual := ruckig.Duration, DELTA := 1E-8, Message := 'Minimum duration not equals duration');

// Check duration for each phase
positionExtrema := ruckig._profiles[0].Bound();
AssertEquals_LREAL(2.0, positionExtrema.Tmax, 1E-9, message:='Profile[0] Tmax incorrect');
AssertEquals_LREAL(414.5353757372092, positionExtrema.Maximum, 1E-9, message:='Profile[0] maximum incorrect');
AssertEquals_LREAL(0.0, positionExtrema.Tmin, 1E-9, message:='Profile[0] Tmin incorrect');
AssertEquals_LREAL(77.60057317918495, positionExtrema.Minimum, 1E-9, message:='Profile[0] minimum incorrect');

positionExtrema := ruckig._profiles[1].Bound();
AssertEquals_LREAL(2.0, positionExtrema.Tmax, 1E-9, message:='Profile[1] Tmax incorrect');
AssertEquals_LREAL(563.6632518811656, positionExtrema.Maximum, 1E-9, message:='Profile[1] maximum incorrect');
AssertEquals_LREAL(0.0, positionExtrema.Tmin, 1E-9, message:='Profile[1] Tmin incorrect');
AssertEquals_LREAL(30.762778737727984, positionExtrema.Minimum, 1E-9, message:='Profile[1] minimum incorrect');

positionExtrema := ruckig._profiles[2].Bound();
AssertEquals_LREAL(1.9999999857302615, positionExtrema.Tmax, 1E-9, message:='Profile[2] Tmax incorrect');
AssertEquals_LREAL(514.7655677601987, positionExtrema.Maximum, 1E-9, message:='Profile[2] maximum incorrect');
AssertEquals_LREAL(0.0, positionExtrema.Tmin, 1E-9, message:='Profile[2] Tmin incorrect');
AssertEquals_LREAL(64.62813070858635, positionExtrema.Minimum, 1E-9, message:='Profile[2] minimum incorrect');
   

TEST_FINISHED();
END_METHOD

METHOD Test_Trajectory_VelIntrf_HasMinDuration_13
VAR_INST

END_VAR
TEST('Trajectory_VelIntrf_HasMinDuration_13');

ruckig();

// Check total duration of profiles
AssertEquals_LREAL(Expected := 1.0, Actual := ruckig.Duration, DELTA := 1E-8, Message := 'Duration incorrect');

// Check minimum duration
AssertEquals_LREAL(Expected := ruckig.MinDuration, Actual := ruckig.Duration, DELTA := 1E-8, Message := 'Minimum duration not equals duration');

// Check duration for each phase
positionExtrema := ruckig._profiles[0].Bound();
AssertEquals_LREAL(1.0, positionExtrema.Tmax, 1E-9, message:='Profile[0] Tmax incorrect');
AssertEquals_LREAL(95.04181868014435, positionExtrema.Maximum, 1E-9, message:='Profile[0] maximum incorrect');
AssertEquals_LREAL(0.0, positionExtrema.Tmin, 1E-9, message:='Profile[0] Tmin incorrect');
AssertEquals_LREAL(84.42864058696819, positionExtrema.Minimum, 1E-9, message:='Profile[0] minimum incorrect');

positionExtrema := ruckig._profiles[1].Bound();
AssertEquals_LREAL(0.0, positionExtrema.Tmax, 1E-9, message:='Profile[1] Tmax incorrect');
AssertEquals_LREAL(-11.7964257097819, positionExtrema.Maximum, 1E-9, message:='Profile[1] maximum incorrect');
AssertEquals_LREAL(0.06154925827901086, positionExtrema.Tmin, 1E-9, message:='Profile[1] Tmin incorrect');
AssertEquals_LREAL(-15.107735508894645, positionExtrema.Minimum, 1E-9, message:='Profile[1] minimum incorrect');

positionExtrema := ruckig._profiles[2].Bound();
AssertEquals_LREAL(0.0, positionExtrema.Tmax, 1E-9, message:='Profile[2] Tmax incorrect');
AssertEquals_LREAL(-59.92935947897627, positionExtrema.Maximum, 1E-9, message:='Profile[2] maximum incorrect');
AssertEquals_LREAL(0.27421715681063157932, positionExtrema.Tmin, 1E-9, message:='Profile[2] Tmin incorrect');
AssertEquals_LREAL(-128.80834180561783, positionExtrema.Minimum, 1E-9, message:='Profile[2] minimum incorrect');
   

TEST_FINISHED();
END_METHOD

METHOD Test_Trajectory_VelIntrf_HasMinDuration_16
VAR_INST
  ruckig : Struckig.Otg(0.001, 3) := (
  
    ControlInterface := ControlInterfaceType.Velocity,
    Synchronization := SynchronizationType.TimeSync,
    MinDuration := 8.0,
    MaxVelocity := [ 2000.0, 2000.0, 2000.0 ],
    MaxAcceleration := [ 20000.0, 20000.0, 20000.0 ],
    MaxJerk := [ 800000.0, 800000.0, 800000.0 ],
    CurrentPosition := [ 16.34026286064214, -10.887974842974131, -6.0946579710083455 ],
    CurrentVelocity := [ -841.771417665662, -815.4357794466523, -729.3097500069106 ],
    CurrentAcceleration := [ 3485.439236026403, 377.6205151850936, -9289.606593644981 ],
    TargetPosition := [ -27.206330261349223, 45.75415534661309, 67.56743756412726 ],
    TargetVelocity := [ 0.0, 0.0, 0.0 ],
    TargetAcceleration := [ 0.0, 0.0, 0.0 ]
  );
  
  positionExtrema : Struckig.ProfileBound;
END_VAR
TEST('Trajectory_VelIntrf_HasMinDuration_16');

ruckig();

// Check total duration of profiles
AssertEquals_LREAL(Expected := 8.0, Actual := ruckig.Duration, DELTA := 1E-8, Message := 'Duration incorrect');

// Check minimum duration
AssertEquals_LREAL(Expected := ruckig.MinDuration, Actual := ruckig.Duration, DELTA := 1E-8, Message := 'Minimum duration not equals duration');

// Check duration for each phase
positionExtrema := ruckig._profiles[0].Bound();
AssertEquals_LREAL(0.0, positionExtrema.Tmax, 1E-9, message:='Profile[0] Tmax incorrect');
AssertEquals_LREAL(16.34026286064214, positionExtrema.Maximum, 1E-9, message:='Profile[0] maximum incorrect');
AssertEquals_LREAL(8.0, positionExtrema.Tmin, 1E-9, message:='Profile[0] Tmin incorrect');
AssertEquals_LREAL(-119.19102824606121, positionExtrema.Minimum, 1E-9, message:='Profile[0] minimum incorrect');

positionExtrema := ruckig._profiles[1].Bound();
AssertEquals_LREAL(0.0, positionExtrema.Tmax, 1E-9, message:='Profile[1] Tmax incorrect');
AssertEquals_LREAL(-10.887974842974131, positionExtrema.Maximum, 1E-9, message:='Profile[1] maximum incorrect');
AssertEquals_LREAL(8.0, positionExtrema.Tmin, 1E-9, message:='Profile[1] Tmin incorrect');
AssertEquals_LREAL(-1184.7922582227166, positionExtrema.Minimum, 1E-9, message:='Profile[1] minimum incorrect');

positionExtrema := ruckig._profiles[2].Bound();
AssertEquals_LREAL(0.0, positionExtrema.Tmax, 1E-9, message:='Profile[2] Tmax incorrect');
AssertEquals_LREAL(-6.0946579710083455, positionExtrema.Maximum, 1E-9, message:='Profile[2] maximum incorrect');
AssertEquals_LREAL(7.9999999738157515, positionExtrema.Tmin, 1E-9, message:='Profile[2] Tmin incorrect');
AssertEquals_LREAL(-3143.4143933071305, positionExtrema.Minimum, 1E-9, message:='Profile[2] minimum incorrect');
   

TEST_FINISHED();
END_METHOD

METHOD Test_Trajectory_VelIntrf_HasMinDuration_18
VAR_INST
  ruckig : Struckig.Otg(0.001, 3) := (
  
    ControlInterface := ControlInterfaceType.Velocity,
    Synchronization := SynchronizationType.TimeSync,
    MinDuration := 6.0,
    MaxVelocity := [ 2000.0, 2000.0, 2000.0 ],
    MaxAcceleration := [ 20000.0, 20000.0, 20000.0 ],
    MaxJerk := [ 800000.0, 800000.0, 800000.0 ],
    CurrentPosition := [ 90.34742980457051, 37.43702634727555, -87.8799213811221 ],
    CurrentVelocity := [ -659.0273208828401, -796.5648287676397, -143.12820706677633 ],
    CurrentAcceleration := [ 8183.9808983774565, 9959.369264181467, 9731.235572560941 ],
    TargetPosition := [ -8.821526080892056, 4.78627195156875, 64.20495391203934 ],
    TargetVelocity := [ 0.0, 0.0, 0.0 ],
    TargetAcceleration := [ 0.0, 0.0, 0.0 ]
  );
  
  positionExtrema : Struckig.ProfileBound;
END_VAR
TEST('Trajectory_VelIntrf_HasMinDuration_18');

ruckig();

// Check total duration of profiles
AssertEquals_LREAL(Expected := 6.0, Actual := ruckig.Duration, DELTA := 1E-8, Message := 'Duration incorrect');

// Check minimum duration
AssertEquals_LREAL(Expected := ruckig.MinDuration, Actual := ruckig.Duration, DELTA := 1E-8, Message := 'Minimum duration not equals duration');

// Check duration for each phase
positionExtrema := ruckig._profiles[0].Bound();
AssertEquals_LREAL(0.0, positionExtrema.Tmax, 1E-9, message:='Profile[0] Tmax incorrect');
AssertEquals_LREAL(90.34742980457051, positionExtrema.Maximum, 1E-9, message:='Profile[0] maximum incorrect');
AssertEquals_LREAL(0.1610529958625631, positionExtrema.Tmin, 1E-9, message:='Profile[0] Tmin incorrect');
AssertEquals_LREAL(54.96798834341715, positionExtrema.Minimum, 1E-9, message:='Profile[0] minimum incorrect');

positionExtrema := ruckig._profiles[1].Bound();
AssertEquals_LREAL(0.0, positionExtrema.Tmax, 1E-9, message:='Profile[1] Tmax incorrect');
AssertEquals_LREAL(37.43702634727555, positionExtrema.Maximum, 1E-9, message:='Profile[1] maximum incorrect');
AssertEquals_LREAL(0.15996290681428152, positionExtrema.Tmin, 1E-9, message:='Profile[1] Tmin incorrect');
AssertEquals_LREAL(-5.0365821446218035, positionExtrema.Minimum, 1E-9, message:='Profile[1] minimum incorrect');

positionExtrema := ruckig._profiles[2].Bound();
AssertEquals_LREAL(0.0, positionExtrema.Tmax, 1E-9, message:='Profile[2] Tmax incorrect');
AssertEquals_LREAL(-87.8799213811221, positionExtrema.Maximum, 1E-9, message:='Profile[2] maximum incorrect');
AssertEquals_LREAL(0.029416245449931017, positionExtrema.Tmin, 1E-9, message:='Profile[2] Tmin incorrect');
AssertEquals_LREAL(-89.28335287108372, positionExtrema.Minimum, 1E-9, message:='Profile[2] minimum incorrect');
   

TEST_FINISHED();
END_METHOD

METHOD Test_Trajectory_VelIntrf_HasMinDuration_27
VAR_INST
  ruckig : Struckig.Otg(0.001, 3) := (
  
    ControlInterface := ControlInterfaceType.Velocity,
    Synchronization := SynchronizationType.TimeSync,
    MinDuration := 3.0,
    MaxVelocity := [ 2000.0, 2000.0, 2000.0 ],
    MaxAcceleration := [ 20000.0, 20000.0, 20000.0 ],
    MaxJerk := [ 800000.0, 800000.0, 800000.0 ],
    CurrentPosition := [ 6.220673442790442, 55.350404818761376, 43.901736472926615 ],
    CurrentVelocity := [ -312.119132016202, 179.9809013069082, -96.87807007344702 ],
    CurrentAcceleration := [ -1455.7993435918852, 6160.858096144148, 3911.3819838930867 ],
    TargetPosition := [ -53.5085757775751, 51.68018231313428, 39.18303391553616 ],
    TargetVelocity := [ 0.0, 0.0, 0.0 ],
    TargetAcceleration := [ 0.0, 0.0, 0.0 ]
  );
  
  positionExtrema : Struckig.ProfileBound;
END_VAR
TEST('Trajectory_VelIntrf_HasMinDuration_27');

ruckig();

// Check total duration of profiles
AssertEquals_LREAL(Expected := 3.0, Actual := ruckig.Duration, DELTA := 1E-8, Message := 'Duration incorrect');

// Check minimum duration
AssertEquals_LREAL(Expected := ruckig.MinDuration, Actual := ruckig.Duration, DELTA := 1E-8, Message := 'Minimum duration not equals duration');

// Check duration for each phase
positionExtrema := ruckig._profiles[0].Bound();
AssertEquals_LREAL(0.0, positionExtrema.Tmax, 1E-9, message:='Profile[0] Tmax incorrect');
AssertEquals_LREAL(6.220673442790442, positionExtrema.Maximum, 1E-9, message:='Profile[0] maximum incorrect');
AssertEquals_LREAL(3.0, positionExtrema.Tmin, 1E-9, message:='Profile[0] Tmin incorrect');
AssertEquals_LREAL(-464.22930783297835, positionExtrema.Minimum, 1E-9, message:='Profile[0] minimum incorrect');

positionExtrema := ruckig._profiles[1].Bound();
AssertEquals_LREAL(2.9999999765561416, positionExtrema.Tmax, 1E-9, message:='Profile[1] Tmax incorrect');
AssertEquals_LREAL(361.6291397294084, positionExtrema.Maximum, 1E-9, message:='Profile[1] maximum incorrect');
AssertEquals_LREAL(0.0, positionExtrema.Tmin, 1E-9, message:='Profile[1] Tmin incorrect');
AssertEquals_LREAL(55.350404818761376, positionExtrema.Minimum, 1E-9, message:='Profile[1] minimum incorrect');

positionExtrema := ruckig._profiles[2].Bound();
AssertEquals_LREAL(0.0, positionExtrema.Tmax, 1E-9, message:='Profile[2] Tmax incorrect');
AssertEquals_LREAL(43.901736472926615, positionExtrema.Maximum, 1E-9, message:='Profile[2] maximum incorrect');
AssertEquals_LREAL(3.0, positionExtrema.Tmin, 1E-9, message:='Profile[2] Tmin incorrect');
AssertEquals_LREAL(42.30206991009092, positionExtrema.Minimum, 1E-9, message:='Profile[2] minimum incorrect');
   

TEST_FINISHED();
END_METHOD

METHOD Test_Trajectory_VelIntrf_HasMinDuration_3
VAR_INST
  ruckig : Struckig.Otg(0.001, 3) := (
  
    ControlInterface := ControlInterfaceType.Velocity,
    Synchronization := SynchronizationType.TimeSync,
    MinDuration := 5.0,
    MaxVelocity := [ 2000.0, 2000.0, 2000.0 ],
    MaxAcceleration := [ 20000.0, 20000.0, 20000.0 ],
    MaxJerk := [ 800000.0, 800000.0, 800000.0 ],
    CurrentPosition := [ -9.67424922051427, 36.41288070877832, -22.139203570767734 ],
    CurrentVelocity := [ -589.9643491179622, -639.1722719741515, 746.8330179980396 ],
    CurrentAcceleration := [ 1695.5266948875524, 4285.3922414822755, -6255.548751889859 ],
    TargetPosition := [ -95.97548318367895, -83.54982092667612, -70.56128130187749 ],
    TargetVelocity := [ 0.0, 0.0, 0.0 ],
    TargetAcceleration := [ 0.0, 0.0, 0.0 ]
  );
  
  positionExtrema : Struckig.ProfileBound;
END_VAR
TEST('Trajectory_VelIntrf_HasMinDuration_3');

ruckig();

// Check total duration of profiles
AssertEquals_LREAL(Expected := 5.0, Actual := ruckig.Duration, DELTA := 1E-8, Message := 'Duration incorrect');

// Check minimum duration
AssertEquals_LREAL(Expected := ruckig.MinDuration, Actual := ruckig.Duration, DELTA := 1E-8, Message := 'Minimum duration not equals duration');

// Check duration for each phase
positionExtrema := ruckig._profiles[0].Bound();
AssertEquals_LREAL(0.0, positionExtrema.Tmax, 1E-9, message:='Profile[0] Tmax incorrect');
AssertEquals_LREAL(-9.67424922051427, positionExtrema.Maximum, 1E-9, message:='Profile[0] maximum incorrect');
AssertEquals_LREAL(5.0, positionExtrema.Tmin, 1E-9, message:='Profile[0] Tmin incorrect');
AssertEquals_LREAL(-146.52766642303507, positionExtrema.Minimum, 1E-9, message:='Profile[0] minimum incorrect');

positionExtrema := ruckig._profiles[1].Bound();
AssertEquals_LREAL(0.0, positionExtrema.Tmax, 1E-9, message:='Profile[1] Tmax incorrect');
AssertEquals_LREAL(36.41288070877832, positionExtrema.Maximum, 1E-9, message:='Profile[1] maximum incorrect');
AssertEquals_LREAL(5.0, positionExtrema.Tmin, 1E-9, message:='Profile[1] Tmin incorrect');
AssertEquals_LREAL(-27.142747378349647, positionExtrema.Minimum, 1E-9, message:='Profile[1] minimum incorrect');

positionExtrema := ruckig._profiles[2].Bound();
AssertEquals_LREAL(5.0, positionExtrema.Tmax, 1E-9, message:='Profile[2] Tmax incorrect');
AssertEquals_LREAL(37.30237689848183, positionExtrema.Maximum, 1E-9, message:='Profile[2] maximum incorrect');
AssertEquals_LREAL(0.0, positionExtrema.Tmin, 1E-9, message:='Profile[2] Tmin incorrect');
AssertEquals_LREAL(-22.139203570767734, positionExtrema.Minimum, 1E-9, message:='Profile[2] minimum incorrect');
   

TEST_FINISHED();
END_METHOD

METHOD Test_Trajectory_VelIntrf_HasMinDuration_30
VAR_INST
  ruckig : Struckig.Otg(0.001, 3) := (
  
    ControlInterface := ControlInterfaceType.Velocity,
    Synchronization := SynchronizationType.TimeSync,
    MinDuration := 3.0,
    MaxVelocity := [ 2000.0, 2000.0, 2000.0 ],
    MaxAcceleration := [ 20000.0, 20000.0, 20000.0 ],
    MaxJerk := [ 800000.0, 800000.0, 800000.0 ],
    CurrentPosition := [ -26.28500599596802, 17.350415040760453, 73.05333099648729 ],
    CurrentVelocity := [ -77.57876275863134, -318.995344872087, -275.87056493527575 ],
    CurrentAcceleration := [ 2926.0610782802487, -3690.9290881003208, 7692.40081125986 ],
    TargetPosition := [ -66.72137259098326, -16.815595700305423, -17.980231379913022 ],
    TargetVelocity := [ 0.0, 0.0, 0.0 ],
    TargetAcceleration := [ 0.0, 0.0, 0.0 ]
  );
  
  positionExtrema : Struckig.ProfileBound;
END_VAR
TEST('Trajectory_VelIntrf_HasMinDuration_30');

ruckig();

// Check total duration of profiles
AssertEquals_LREAL(Expected := 3.0, Actual := ruckig.Duration, DELTA := 1E-8, Message := 'Duration incorrect');

// Check minimum duration
AssertEquals_LREAL(Expected := ruckig.MinDuration, Actual := ruckig.Duration, DELTA := 1E-8, Message := 'Minimum duration not equals duration');

// Check duration for each phase
positionExtrema := ruckig._profiles[0].Bound();
AssertEquals_LREAL(0.0, positionExtrema.Tmax, 1E-9, message:='Profile[0] Tmax incorrect');
AssertEquals_LREAL(-26.28500599596802, positionExtrema.Maximum, 1E-9, message:='Profile[0] maximum incorrect');
AssertEquals_LREAL(0.05302607203553466, positionExtrema.Tmin, 1E-9, message:='Profile[0] Tmin incorrect');
AssertEquals_LREAL(-27.656238350123633, positionExtrema.Minimum, 1E-9, message:='Profile[0] minimum incorrect');

positionExtrema := ruckig._profiles[1].Bound();
AssertEquals_LREAL(0.0, positionExtrema.Tmax, 1E-9, message:='Profile[1] Tmax incorrect');
AssertEquals_LREAL(17.350415040760453, positionExtrema.Maximum, 1E-9, message:='Profile[1] maximum incorrect');
AssertEquals_LREAL(2.9999999739834657, positionExtrema.Tmin, 1E-9, message:='Profile[1] Tmin incorrect');
AssertEquals_LREAL(-474.65654025627595, positionExtrema.Minimum, 1E-9, message:='Profile[1] minimum incorrect');

positionExtrema := ruckig._profiles[2].Bound();
AssertEquals_LREAL(0.0, positionExtrema.Tmax, 1E-9, message:='Profile[2] Tmax incorrect');
AssertEquals_LREAL(73.05333099648729, positionExtrema.Maximum, 1E-9, message:='Profile[2] maximum incorrect');
AssertEquals_LREAL(0.07172547861298811, positionExtrema.Tmin, 1E-9, message:='Profile[2] Tmin incorrect');
AssertEquals_LREAL(66.4576815614146, positionExtrema.Minimum, 1E-9, message:='Profile[2] minimum incorrect');
   

TEST_FINISHED();
END_METHOD

METHOD Test_Trajectory_VelIntrf_HasMinDuration_32
VAR_INST
  ruckig : Struckig.Otg(0.001, 3) := (
  
    ControlInterface := ControlInterfaceType.Velocity,
    Synchronization := SynchronizationType.TimeSync,
    MinDuration := 4.0,
    MaxVelocity := [ 2000.0, 2000.0, 2000.0 ],
    MaxAcceleration := [ 20000.0, 20000.0, 20000.0 ],
    MaxJerk := [ 800000.0, 800000.0, 800000.0 ],
    CurrentPosition := [ 12.929925233306733, 54.78105812816395, 9.633021170337713 ],
    CurrentVelocity := [ 690.6885698507674, 500.03919079149, 740.0977409308255 ],
    CurrentAcceleration := [ -6082.612459119506, -7695.992942287852, -8226.103496487962 ],
    TargetPosition := [ 0.5083043656089785, -60.84677752217185, -49.14840333769259 ],
    TargetVelocity := [ 0.0, 0.0, 0.0 ],
    TargetAcceleration := [ 0.0, 0.0, 0.0 ]
  );
  
  positionExtrema : Struckig.ProfileBound;
END_VAR
TEST('Trajectory_VelIntrf_HasMinDuration_32');

ruckig();

// Check total duration of profiles
AssertEquals_LREAL(Expected := 4.0, Actual := ruckig.Duration, DELTA := 1E-8, Message := 'Duration incorrect');

// Check minimum duration
AssertEquals_LREAL(Expected := ruckig.MinDuration, Actual := ruckig.Duration, DELTA := 1E-8, Message := 'Minimum duration not equals duration');

// Check duration for each phase
positionExtrema := ruckig._profiles[0].Bound();
AssertEquals_LREAL(4.0, positionExtrema.Tmax, 1E-9, message:='Profile[0] Tmax incorrect');
AssertEquals_LREAL(65.21564990931404, positionExtrema.Maximum, 1E-9, message:='Profile[0] maximum incorrect');
AssertEquals_LREAL(0.0, positionExtrema.Tmin, 1E-9, message:='Profile[0] Tmin incorrect');
AssertEquals_LREAL(12.929925233306733, positionExtrema.Minimum, 1E-9, message:='Profile[0] minimum incorrect');

positionExtrema := ruckig._profiles[1].Bound();
AssertEquals_LREAL(0.1299479338251158, positionExtrema.Tmax, 1E-9, message:='Profile[1] Tmax incorrect');
AssertEquals_LREAL(76.44074468647628, positionExtrema.Maximum, 1E-9, message:='Profile[1] maximum incorrect');
AssertEquals_LREAL(0.0, positionExtrema.Tmin, 1E-9, message:='Profile[1] Tmin incorrect');
AssertEquals_LREAL(54.78105812816395, positionExtrema.Minimum, 1E-9, message:='Profile[1] minimum incorrect');

positionExtrema := ruckig._profiles[2].Bound();
AssertEquals_LREAL(0.17993883525700874, positionExtrema.Tmax, 1E-9, message:='Profile[2] Tmax incorrect');
AssertEquals_LREAL(54.02379633014975, positionExtrema.Maximum, 1E-9, message:='Profile[2] maximum incorrect');
AssertEquals_LREAL(0.0, positionExtrema.Tmin, 1E-9, message:='Profile[2] Tmin incorrect');
AssertEquals_LREAL(9.633021170337713, positionExtrema.Minimum, 1E-9, message:='Profile[2] minimum incorrect');
   

TEST_FINISHED();
END_METHOD

METHOD Test_Trajectory_VelIntrf_HasMinDuration_34
VAR_INST
  ruckig : Struckig.Otg(0.001, 3) := (
  
    ControlInterface := ControlInterfaceType.Velocity,
    Synchronization := SynchronizationType.TimeSync,
    MinDuration := 1.0,
    MaxVelocity := [ 2000.0, 2000.0, 2000.0 ],
    MaxAcceleration := [ 20000.0, 20000.0, 20000.0 ],
    MaxJerk := [ 800000.0, 800000.0, 800000.0 ],
    CurrentPosition := [ 52.27373667705652, 42.38008848555776, -16.663069900943682 ],
    CurrentVelocity := [ -593.7282384512066, 598.7500512251315, -361.8583055849782 ],
    CurrentAcceleration := [ -6262.0050324295535, 4603.582350239803, -8651.94800823453 ],
    TargetPosition := [ -16.307807021664388, -73.89058906441932, -94.85216176897013 ],
    TargetVelocity := [ 0.0, 0.0, 0.0 ],
    TargetAcceleration := [ 0.0, 0.0, 0.0 ]
  );
  
  positionExtrema : Struckig.ProfileBound;
END_VAR
TEST('Trajectory_VelIntrf_HasMinDuration_34');

ruckig();

// Check total duration of profiles
AssertEquals_LREAL(Expected := 1.0, Actual := ruckig.Duration, DELTA := 1E-8, Message := 'Duration incorrect');

// Check minimum duration
AssertEquals_LREAL(Expected := ruckig.MinDuration, Actual := ruckig.Duration, DELTA := 1E-8, Message := 'Minimum duration not equals duration');

// Check duration for each phase
positionExtrema := ruckig._profiles[0].Bound();
AssertEquals_LREAL(0.0, positionExtrema.Tmax, 1E-9, message:='Profile[0] Tmax incorrect');
AssertEquals_LREAL(52.27373667705652, positionExtrema.Maximum, 1E-9, message:='Profile[0] maximum incorrect');
AssertEquals_LREAL(1.0, positionExtrema.Tmin, 1E-9, message:='Profile[0] Tmin incorrect');
AssertEquals_LREAL(-259.2000319331284, positionExtrema.Minimum, 1E-9, message:='Profile[0] minimum incorrect');

positionExtrema := ruckig._profiles[1].Bound();
AssertEquals_LREAL(1.0, positionExtrema.Tmax, 1E-9, message:='Profile[1] Tmax incorrect');
AssertEquals_LREAL(350.1133679372294, positionExtrema.Maximum, 1E-9, message:='Profile[1] maximum incorrect');
AssertEquals_LREAL(0.0, positionExtrema.Tmin, 1E-9, message:='Profile[1] Tmin incorrect');
AssertEquals_LREAL(42.38008848555776, positionExtrema.Minimum, 1E-9, message:='Profile[1] minimum incorrect');

positionExtrema := ruckig._profiles[2].Bound();
AssertEquals_LREAL(0.0, positionExtrema.Tmax, 1E-9, message:='Profile[2] Tmax incorrect');
AssertEquals_LREAL(-16.663069900943682, positionExtrema.Maximum, 1E-9, message:='Profile[2] maximum incorrect');
AssertEquals_LREAL(1.0, positionExtrema.Tmin, 1E-9, message:='Profile[2] Tmin incorrect');
AssertEquals_LREAL(-223.02585326367077, positionExtrema.Minimum, 1E-9, message:='Profile[2] minimum incorrect');
   

TEST_FINISHED();
END_METHOD

METHOD Test_Trajectory_VelIntrf_HasMinDuration_36
VAR_INST
  ruckig : Struckig.Otg(0.001, 3) := (
  
    ControlInterface := ControlInterfaceType.Velocity,
    Synchronization := SynchronizationType.TimeSync,
    MinDuration := 3.0,
    MaxVelocity := [ 2000.0, 2000.0, 2000.0 ],
    MaxAcceleration := [ 20000.0, 20000.0, 20000.0 ],
    MaxJerk := [ 800000.0, 800000.0, 800000.0 ],
    CurrentPosition := [ 89.58406345666467, -82.12124040809996, 44.15238439970966 ],
    CurrentVelocity := [ 860.6527066721621, -645.8300161653469, -25.24004639866348 ],
    CurrentAcceleration := [ 100.52505589197972, 9013.944448759463, 5339.978050227286 ],
    TargetPosition := [ 69.92494471362522, -54.90917502215438, -64.642348891492 ],
    TargetVelocity := [ 0.0, 0.0, 0.0 ],
    TargetAcceleration := [ 0.0, 0.0, 0.0 ]
  );
  
  positionExtrema : Struckig.ProfileBound;
END_VAR
TEST('Trajectory_VelIntrf_HasMinDuration_36');

ruckig();

// Check total duration of profiles
AssertEquals_LREAL(Expected := 3.0, Actual := ruckig.Duration, DELTA := 1E-8, Message := 'Duration incorrect');

// Check minimum duration
AssertEquals_LREAL(Expected := ruckig.MinDuration, Actual := ruckig.Duration, DELTA := 1E-8, Message := 'Minimum duration not equals duration');

// Check duration for each phase
positionExtrema := ruckig._profiles[0].Bound();
AssertEquals_LREAL(2.9999999768762042, positionExtrema.Tmax, 1E-9, message:='Profile[0] Tmax incorrect');
AssertEquals_LREAL(1380.6266705291914, positionExtrema.Maximum, 1E-9, message:='Profile[0] maximum incorrect');
AssertEquals_LREAL(0.0, positionExtrema.Tmin, 1E-9, message:='Profile[0] Tmin incorrect');
AssertEquals_LREAL(89.58406345666467, positionExtrema.Minimum, 1E-9, message:='Profile[0] minimum incorrect');

positionExtrema := ruckig._profiles[1].Bound();
AssertEquals_LREAL(0.0, positionExtrema.Tmax, 1E-9, message:='Profile[1] Tmax incorrect');
AssertEquals_LREAL(-82.12124040809996, positionExtrema.Maximum, 1E-9, message:='Profile[1] maximum incorrect');
AssertEquals_LREAL(3.0, positionExtrema.Tmin, 1E-9, message:='Profile[1] Tmin incorrect');
AssertEquals_LREAL(-112.96947502586413, positionExtrema.Minimum, 1E-9, message:='Profile[1] minimum incorrect');

positionExtrema := ruckig._profiles[2].Bound();
AssertEquals_LREAL(0.0, positionExtrema.Tmax, 1E-9, message:='Profile[2] Tmax incorrect');
AssertEquals_LREAL(44.15238439970966, positionExtrema.Maximum, 1E-9, message:='Profile[2] maximum incorrect');
AssertEquals_LREAL(3.0, positionExtrema.Tmin, 1E-9, message:='Profile[2] Tmin incorrect');
AssertEquals_LREAL(44.07285099636173, positionExtrema.Minimum, 1E-9, message:='Profile[2] minimum incorrect');
   

TEST_FINISHED();
END_METHOD

METHOD Test_Trajectory_VelIntrf_HasMinDuration_38
VAR_INST
  ruckig : Struckig.Otg(0.001, 3) := (
  
    ControlInterface := ControlInterfaceType.Velocity,
    Synchronization := SynchronizationType.TimeSync,
    MinDuration := 3.0,
    MaxVelocity := [ 2000.0, 2000.0, 2000.0 ],
    MaxAcceleration := [ 20000.0, 20000.0, 20000.0 ],
    MaxJerk := [ 800000.0, 800000.0, 800000.0 ],
    CurrentPosition := [ 37.307673430642495, -93.34690301601272, -11.774723734847896 ],
    CurrentVelocity := [ -121.25389830691358, -668.1202626334424, 122.25742950217364 ],
    CurrentAcceleration := [ -3440.0239449720284, 226.88867779635257, -9737.166378946953 ],
    TargetPosition := [ 34.34181137247978, 99.7596266578339, 54.67868464456106 ],
    TargetVelocity := [ 0.0, 0.0, 0.0 ],
    TargetAcceleration := [ 0.0, 0.0, 0.0 ]
  );
  
  positionExtrema : Struckig.ProfileBound;
END_VAR
TEST('Trajectory_VelIntrf_HasMinDuration_38');

ruckig();

// Check total duration of profiles
AssertEquals_LREAL(Expected := 3.0, Actual := ruckig.Duration, DELTA := 1E-8, Message := 'Duration incorrect');

// Check minimum duration
AssertEquals_LREAL(Expected := ruckig.MinDuration, Actual := ruckig.Duration, DELTA := 1E-8, Message := 'Minimum duration not equals duration');

// Check duration for each phase
positionExtrema := ruckig._profiles[0].Bound();
AssertEquals_LREAL(0.0, positionExtrema.Tmax, 1E-9, message:='Profile[0] Tmax incorrect');
AssertEquals_LREAL(37.307673430642495, positionExtrema.Maximum, 1E-9, message:='Profile[0] maximum incorrect');
AssertEquals_LREAL(3.0, positionExtrema.Tmin, 1E-9, message:='Profile[0] Tmin incorrect');
AssertEquals_LREAL(-155.93332674897468, positionExtrema.Minimum, 1E-9, message:='Profile[0] minimum incorrect');

positionExtrema := ruckig._profiles[1].Bound();
AssertEquals_LREAL(0.0, positionExtrema.Tmax, 1E-9, message:='Profile[1] Tmax incorrect');
AssertEquals_LREAL(-93.34690301601272, positionExtrema.Maximum, 1E-9, message:='Profile[1] maximum incorrect');
AssertEquals_LREAL(2.9999999996791167, positionExtrema.Tmin, 1E-9, message:='Profile[1] Tmin incorrect');
AssertEquals_LREAL(-1095.4807808100672, positionExtrema.Minimum, 1E-9, message:='Profile[1] minimum incorrect');

positionExtrema := ruckig._profiles[2].Bound();
AssertEquals_LREAL(0.02511150056273259, positionExtrema.Tmax, 1E-9, message:='Profile[2] Tmax incorrect');
AssertEquals_LREAL(-10.751367898267205, positionExtrema.Maximum, 1E-9, message:='Profile[2] maximum incorrect');
AssertEquals_LREAL(0.0, positionExtrema.Tmin, 1E-9, message:='Profile[2] Tmin incorrect');
AssertEquals_LREAL(-11.774723734847896, positionExtrema.Minimum, 1E-9, message:='Profile[2] minimum incorrect');
   

TEST_FINISHED();
END_METHOD

METHOD Test_Trajectory_VelIntrf_HasMinDuration_39
VAR_INST
  ruckig : Struckig.Otg(0.001, 3) := (
  
    ControlInterface := ControlInterfaceType.Velocity,
    Synchronization := SynchronizationType.TimeSync,
    MinDuration := 2.0,
    MaxVelocity := [ 2000.0, 2000.0, 2000.0 ],
    MaxAcceleration := [ 20000.0, 20000.0, 20000.0 ],
    MaxJerk := [ 800000.0, 800000.0, 800000.0 ],
    CurrentPosition := [ -20.616254291671538, -90.11547835294334, -93.95803295464518 ],
    CurrentVelocity := [ 783.0566484103024, 147.8098644695658, 269.1213449142149 ],
    CurrentAcceleration := [ 8600.93347684592, -8314.610641760264, -9302.258281844754 ],
    TargetPosition := [ 90.57210220298848, 11.32679444144837, 40.182871392763275 ],
    TargetVelocity := [ 0.0, 0.0, 0.0 ],
    TargetAcceleration := [ 0.0, 0.0, 0.0 ]
  );
  
  positionExtrema : Struckig.ProfileBound;
END_VAR
TEST('Trajectory_VelIntrf_HasMinDuration_39');

ruckig();

// Check total duration of profiles
AssertEquals_LREAL(Expected := 2.0, Actual := ruckig.Duration, DELTA := 1E-8, Message := 'Duration incorrect');

// Check minimum duration
AssertEquals_LREAL(Expected := ruckig.MinDuration, Actual := ruckig.Duration, DELTA := 1E-8, Message := 'Minimum duration not equals duration');

// Check duration for each phase
positionExtrema := ruckig._profiles[0].Bound();
AssertEquals_LREAL(2.0, positionExtrema.Tmax, 1E-9, message:='Profile[0] Tmax incorrect');
AssertEquals_LREAL(812.9676626411957, positionExtrema.Maximum, 1E-9, message:='Profile[0] maximum incorrect');
AssertEquals_LREAL(0.0, positionExtrema.Tmin, 1E-9, message:='Profile[0] Tmin incorrect');
AssertEquals_LREAL(-20.616254291671538, positionExtrema.Minimum, 1E-9, message:='Profile[0] minimum incorrect');

positionExtrema := ruckig._profiles[1].Bound();
AssertEquals_LREAL(0.035554248019068604, positionExtrema.Tmax, 1E-9, message:='Profile[1] Tmax incorrect');
AssertEquals_LREAL(-88.36372215927139, positionExtrema.Maximum, 1E-9, message:='Profile[1] maximum incorrect');
AssertEquals_LREAL(0.0, positionExtrema.Tmin, 1E-9, message:='Profile[1] Tmin incorrect');
AssertEquals_LREAL(-90.11547835294334, positionExtrema.Minimum, 1E-9, message:='Profile[1] minimum incorrect');

positionExtrema := ruckig._profiles[2].Bound();
AssertEquals_LREAL(0.05786150776730417, positionExtrema.Tmax, 1E-9, message:='Profile[2] Tmax incorrect');
AssertEquals_LREAL(-88.76744402494478, positionExtrema.Maximum, 1E-9, message:='Profile[2] maximum incorrect');
AssertEquals_LREAL(0.0, positionExtrema.Tmin, 1E-9, message:='Profile[2] Tmin incorrect');
AssertEquals_LREAL(-93.95803295464518, positionExtrema.Minimum, 1E-9, message:='Profile[2] minimum incorrect');
   

TEST_FINISHED();
END_METHOD

METHOD Test_Trajectory_VelIntrf_HasMinDuration_4
VAR_INST
  ruckig : Struckig.Otg(0.001, 3) := (
  
    ControlInterface := ControlInterfaceType.Velocity,
    Synchronization := SynchronizationType.TimeSync,
    MinDuration := 9.0,
    MaxVelocity := [ 2000.0, 2000.0, 2000.0 ],
    MaxAcceleration := [ 20000.0, 20000.0, 20000.0 ],
    MaxJerk := [ 800000.0, 800000.0, 800000.0 ],
    CurrentPosition := [ 62.02540605044314, -71.46568692377213, -39.17183777062583 ],
    CurrentVelocity := [ 852.1519572293494, -167.96910985910404, 848.0360997635792 ],
    CurrentAcceleration := [ -5929.687089686932, 6537.284294646994, -5825.200057211235 ],
    TargetPosition := [ -33.09491825100352, -50.62227338441654, -22.42151000841966 ],
    TargetVelocity := [ 0.0, 0.0, 0.0 ],
    TargetAcceleration := [ 0.0, 0.0, 0.0 ]
  );
  
  positionExtrema : Struckig.ProfileBound;
END_VAR
TEST('Trajectory_VelIntrf_HasMinDuration_4');

ruckig();

// Check total duration of profiles
AssertEquals_LREAL(Expected := 9.0, Actual := ruckig.Duration, DELTA := 1E-8, Message := 'Duration incorrect');

// Check minimum duration
AssertEquals_LREAL(Expected := ruckig.MinDuration, Actual := ruckig.Duration, DELTA := 1E-8, Message := 'Minimum duration not equals duration');

// Check duration for each phase
positionExtrema := ruckig._profiles[0].Bound();
AssertEquals_LREAL(0.2874188618524018, positionExtrema.Tmax, 1E-9, message:='Profile[0] Tmax incorrect');
AssertEquals_LREAL(143.66692127449517, positionExtrema.Maximum, 1E-9, message:='Profile[0] maximum incorrect');
AssertEquals_LREAL(0.0, positionExtrema.Tmin, 1E-9, message:='Profile[0] Tmin incorrect');
AssertEquals_LREAL(62.02540605044314, positionExtrema.Minimum, 1E-9, message:='Profile[0] minimum incorrect');

positionExtrema := ruckig._profiles[1].Bound();
AssertEquals_LREAL(0.0, positionExtrema.Tmax, 1E-9, message:='Profile[1] Tmax incorrect');
AssertEquals_LREAL(-71.46568692377213, positionExtrema.Maximum, 1E-9, message:='Profile[1] maximum incorrect');
AssertEquals_LREAL(9.0, positionExtrema.Tmin, 1E-9, message:='Profile[1] Tmin incorrect');
AssertEquals_LREAL(-74.34288797501209, positionExtrema.Minimum, 1E-9, message:='Profile[1] minimum incorrect');

positionExtrema := ruckig._profiles[2].Bound();
AssertEquals_LREAL(0.29116119324134226, positionExtrema.Tmax, 1E-9, message:='Profile[2] Tmax incorrect');
AssertEquals_LREAL(43.133229802340054, positionExtrema.Maximum, 1E-9, message:='Profile[2] maximum incorrect');
AssertEquals_LREAL(0.0, positionExtrema.Tmin, 1E-9, message:='Profile[2] Tmin incorrect');
AssertEquals_LREAL(-39.17183777062583, positionExtrema.Minimum, 1E-9, message:='Profile[2] minimum incorrect');
   

TEST_FINISHED();
END_METHOD

METHOD Test_Trajectory_VelIntrf_HasMinDuration_6
VAR_INST
  ruckig : Struckig.Otg(0.001, 3) := (
  
    ControlInterface := ControlInterfaceType.Velocity,
    Synchronization := SynchronizationType.TimeSync,
    MinDuration := 4.0,
    MaxVelocity := [ 2000.0, 2000.0, 2000.0 ],
    MaxAcceleration := [ 20000.0, 20000.0, 20000.0 ],
    MaxJerk := [ 800000.0, 800000.0, 800000.0 ],
    CurrentPosition := [ -95.48128756599684, -11.887604170884302, 13.304818742686166 ],
    CurrentVelocity := [ 742.9483502145449, -75.8918641984609, -212.06650304832044 ],
    CurrentAcceleration := [ -5422.793382334212, 5015.348084009836, 5723.627908682256 ],
    TargetPosition := [ 87.51986212872634, -16.94845049603282, 71.8626135805398 ],
    TargetVelocity := [ 0.0, 0.0, 0.0 ],
    TargetAcceleration := [ 0.0, 0.0, 0.0 ]
  );
  
  positionExtrema : Struckig.ProfileBound;
END_VAR
TEST('Trajectory_VelIntrf_HasMinDuration_6');

ruckig();

// Check total duration of profiles
AssertEquals_LREAL(Expected := 4.0, Actual := ruckig.Duration, DELTA := 1E-8, Message := 'Duration incorrect');

// Check minimum duration
AssertEquals_LREAL(Expected := ruckig.MinDuration, Actual := ruckig.Duration, DELTA := 1E-8, Message := 'Minimum duration not equals duration');

// Check duration for each phase
positionExtrema := ruckig._profiles[0].Bound();
AssertEquals_LREAL(4.0, positionExtrema.Tmax, 1E-9, message:='Profile[0] Tmax incorrect');
AssertEquals_LREAL(-27.62299484122707, positionExtrema.Maximum, 1E-9, message:='Profile[0] maximum incorrect');
AssertEquals_LREAL(0.0, positionExtrema.Tmin, 1E-9, message:='Profile[0] Tmin incorrect');
AssertEquals_LREAL(-95.48128756599684, positionExtrema.Minimum, 1E-9, message:='Profile[0] minimum incorrect');

positionExtrema := ruckig._profiles[1].Bound();
AssertEquals_LREAL(0.0, positionExtrema.Tmax, 1E-9, message:='Profile[1] Tmax incorrect');
AssertEquals_LREAL(-11.887604170884302, positionExtrema.Maximum, 1E-9, message:='Profile[1] maximum incorrect');
AssertEquals_LREAL(0.030263846897025354, positionExtrema.Tmin, 1E-9, message:='Profile[1] Tmin incorrect');
AssertEquals_LREAL(-12.653197433145344, positionExtrema.Minimum, 1E-9, message:='Profile[1] minimum incorrect');

positionExtrema := ruckig._profiles[2].Bound();
AssertEquals_LREAL(0.0, positionExtrema.Tmax, 1E-9, message:='Profile[2] Tmax incorrect');
AssertEquals_LREAL(13.304818742686166, positionExtrema.Maximum, 1E-9, message:='Profile[2] maximum incorrect');
AssertEquals_LREAL(4.0, positionExtrema.Tmin, 1E-9, message:='Profile[2] Tmin incorrect');
AssertEquals_LREAL(8.066625713985442, positionExtrema.Minimum, 1E-9, message:='Profile[2] minimum incorrect');
   

TEST_FINISHED();
END_METHOD

METHOD Test_Trajectory_VelIntrf_HasMinDuration_8
VAR_INST
  ruckig : Struckig.Otg(0.001, 3) := (
  
    ControlInterface := ControlInterfaceType.Velocity,
    Synchronization := SynchronizationType.TimeSync,
    MinDuration := 4.0,
    MaxVelocity := [ 2000.0, 2000.0, 2000.0 ],
    MaxAcceleration := [ 20000.0, 20000.0, 20000.0 ],
    MaxJerk := [ 800000.0, 800000.0, 800000.0 ],
    CurrentPosition := [ 13.23871132942243, 76.70197428551197, -81.05183127225158 ],
    CurrentVelocity := [ -435.93783540226855, 450.149281088266, -270.1461541941925 ],
    CurrentAcceleration := [ 758.8421967400063, -6759.552729506426, 1610.794729644338 ],
    TargetPosition := [ -97.66489958402742, 89.83230792788837, 24.731322190695778 ],
    TargetVelocity := [ 0.0, 0.0, 0.0 ],
    TargetAcceleration := [ 0.0, 0.0, 0.0 ]
  );
  
  positionExtrema : Struckig.ProfileBound;
END_VAR
TEST('Trajectory_VelIntrf_HasMinDuration_8');

ruckig();

// Check total duration of profiles
AssertEquals_LREAL(Expected := 4.0, Actual := ruckig.Duration, DELTA := 1E-8, Message := 'Duration incorrect');

// Check minimum duration
AssertEquals_LREAL(Expected := ruckig.MinDuration, Actual := ruckig.Duration, DELTA := 1E-8, Message := 'Minimum duration not equals duration');

// Check duration for each phase
positionExtrema := ruckig._profiles[0].Bound();
AssertEquals_LREAL(0.0, positionExtrema.Tmax, 1E-9, message:='Profile[0] Tmax incorrect');
AssertEquals_LREAL(13.23871132942243, positionExtrema.Maximum, 1E-9, message:='Profile[0] maximum incorrect');
AssertEquals_LREAL(1.1489551774402158, positionExtrema.Tmin, 1E-9, message:='Profile[0] Tmin incorrect');
AssertEquals_LREAL(-153.71896634641655, positionExtrema.Minimum, 1E-9, message:='Profile[0] minimum incorrect');

positionExtrema := ruckig._profiles[1].Bound();
AssertEquals_LREAL(4.0, positionExtrema.Tmax, 1E-9, message:='Profile[1] Tmax incorrect');
AssertEquals_LREAL(96.68696277741057, positionExtrema.Maximum, 1E-9, message:='Profile[1] maximum incorrect');
AssertEquals_LREAL(0.0, positionExtrema.Tmin, 1E-9, message:='Profile[1] Tmin incorrect');
AssertEquals_LREAL(76.70197428551197, positionExtrema.Minimum, 1E-9, message:='Profile[1] minimum incorrect');

positionExtrema := ruckig._profiles[2].Bound();
AssertEquals_LREAL(0.0, positionExtrema.Tmax, 1E-9, message:='Profile[2] Tmax incorrect');
AssertEquals_LREAL(-81.05183127225158, positionExtrema.Maximum, 1E-9, message:='Profile[2] maximum incorrect');
AssertEquals_LREAL(0.3354197145328884, positionExtrema.Tmin, 1E-9, message:='Profile[2] Tmin incorrect');
AssertEquals_LREAL(-111.25594657957613, positionExtrema.Minimum, 1E-9, message:='Profile[2] minimum incorrect');
   

TEST_FINISHED();
END_METHOD

METHOD Test_Trajectory_VelIntrf_HasMinDuration_HasTargetAcceleration_12
VAR_INST
  ruckig : Struckig.Otg(0.001, 3) := (
  
    ControlInterface := ControlInterfaceType.Velocity,
    Synchronization := SynchronizationType.TimeSync,
    MinDuration := 2.0,
    MaxVelocity := [ 2000.0, 2000.0, 2000.0 ],
    MaxAcceleration := [ 20000.0, 20000.0, 20000.0 ],
    MaxJerk := [ 800000.0, 800000.0, 800000.0 ],
    CurrentPosition := [ -43.48377042985394, 17.3008509790114, 62.92824674049976 ],
    CurrentVelocity := [ -465.33252136556587, 82.11778677897496, 322.8916761532398 ],
    CurrentAcceleration := [ 6251.275546033887, -1224.8767937973225, -9034.04310260991 ],
    TargetPosition := [ -79.21888060660451, -54.145883802865555, -86.80139306063326 ],
    TargetVelocity := [ 0.0, 0.0, 0.0 ],
    TargetAcceleration := [ -944.4260728155158, -461.14473822234197, -228.97757502312402 ]
  );
  
  positionExtrema : Struckig.ProfileBound;
END_VAR
TEST('Trajectory_VelIntrf_HasMinDuration_HasTargetAcceleration_12');

ruckig();

// Check total duration of profiles
AssertEquals_LREAL(Expected := 2.0, Actual := ruckig.Duration, DELTA := 1E-8, Message := 'Duration incorrect');

// Check minimum duration
AssertEquals_LREAL(Expected := ruckig.MinDuration, Actual := ruckig.Duration, DELTA := 1E-8, Message := 'Minimum duration not equals duration');

// Check duration for each phase
positionExtrema := ruckig._profiles[0].Bound();
AssertEquals_LREAL(2.0, positionExtrema.Tmax, 1E-9, message:='Profile[0] Tmax incorrect');
AssertEquals_LREAL(1331.89651474086, positionExtrema.Maximum, 1E-9, message:='Profile[0] maximum incorrect');
AssertEquals_LREAL(0.08007838326290945, positionExtrema.Tmin, 1E-9, message:='Profile[0] Tmin incorrect');
AssertEquals_LREAL(-61.64472089659309, positionExtrema.Minimum, 1E-9, message:='Profile[0] minimum incorrect');

positionExtrema := ruckig._profiles[1].Bound();
AssertEquals_LREAL(1.9999999999999885, positionExtrema.Tmax, 1E-9, message:='Profile[1] Tmax incorrect');
AssertEquals_LREAL(98.65298431327531, positionExtrema.Maximum, 1E-9, message:='Profile[1] maximum incorrect');
AssertEquals_LREAL(0.0, positionExtrema.Tmin, 1E-9, message:='Profile[1] Tmin incorrect');
AssertEquals_LREAL(17.3008509790114, positionExtrema.Minimum, 1E-9, message:='Profile[1] minimum incorrect');

positionExtrema := ruckig._profiles[2].Bound();
AssertEquals_LREAL(2.0, positionExtrema.Tmax, 1E-9, message:='Profile[2] Tmax incorrect');
AssertEquals_LREAL(336.5320226880611, positionExtrema.Maximum, 1E-9, message:='Profile[2] maximum incorrect');
AssertEquals_LREAL(0.0, positionExtrema.Tmin, 1E-9, message:='Profile[2] Tmin incorrect');
AssertEquals_LREAL(62.92824674049976, positionExtrema.Minimum, 1E-9, message:='Profile[2] minimum incorrect');
   

TEST_FINISHED();
END_METHOD

METHOD Test_Trajectory_VelIntrf_HasMinDuration_HasTargetAcceleration_14
VAR_INST
  ruckig : Struckig.Otg(0.001, 3) := (
  
    ControlInterface := ControlInterfaceType.Velocity,
    Synchronization := SynchronizationType.TimeSync,
    MinDuration := 4.0,
    MaxVelocity := [ 2000.0, 2000.0, 2000.0 ],
    MaxAcceleration := [ 20000.0, 20000.0, 20000.0 ],
    MaxJerk := [ 800000.0, 800000.0, 800000.0 ],
    CurrentPosition := [ -85.85647725852267, -18.469753286611606, 64.22798249457017 ],
    CurrentVelocity := [ -991.4537367187979, 605.03210452653, -255.638165301316 ],
    CurrentAcceleration := [ -899.1512815539736, -9674.478997725528, 5794.543535027777 ],
    TargetPosition := [ 90.36951082423775, -37.7110342068234, -27.45853535617691 ],
    TargetVelocity := [ 0.0, 0.0, 0.0 ],
    TargetAcceleration := [ -181.55119129292507, 720.5104054661081, -310.4205198639978 ]
  );
  
  positionExtrema : Struckig.ProfileBound;
END_VAR
TEST('Trajectory_VelIntrf_HasMinDuration_HasTargetAcceleration_14');

ruckig();

// Check total duration of profiles
AssertEquals_LREAL(Expected := 4.0, Actual := ruckig.Duration, DELTA := 1E-8, Message := 'Duration incorrect');

// Check minimum duration
AssertEquals_LREAL(Expected := ruckig.MinDuration, Actual := ruckig.Duration, DELTA := 1E-8, Message := 'Minimum duration not equals duration');

// Check duration for each phase
positionExtrema := ruckig._profiles[0].Bound();
AssertEquals_LREAL(0.0, positionExtrema.Tmax, 1E-9, message:='Profile[0] Tmax incorrect');
AssertEquals_LREAL(-85.85647725852267, positionExtrema.Maximum, 1E-9, message:='Profile[0] maximum incorrect');
AssertEquals_LREAL(3.999546122022509, positionExtrema.Tmin, 1E-9, message:='Profile[0] Tmin incorrect');
AssertEquals_LREAL(-2070.178062342364, positionExtrema.Minimum, 1E-9, message:='Profile[0] minimum incorrect');

positionExtrema := ruckig._profiles[1].Bound();
AssertEquals_LREAL(0.06603027302284342, positionExtrema.Tmax, 1E-9, message:='Profile[1] Tmax incorrect');
AssertEquals_LREAL(1.1337535837276427, positionExtrema.Maximum, 1E-9, message:='Profile[1] maximum incorrect');
AssertEquals_LREAL(4.0, positionExtrema.Tmin, 1E-9, message:='Profile[1] Tmin incorrect');
AssertEquals_LREAL(-5002.710408011158, positionExtrema.Minimum, 1E-9, message:='Profile[1] minimum incorrect');

positionExtrema := ruckig._profiles[2].Bound();
AssertEquals_LREAL(4.0, positionExtrema.Tmax, 1E-9, message:='Profile[2] Tmax incorrect');
AssertEquals_LREAL(2302.767558744343, positionExtrema.Maximum, 1E-9, message:='Profile[2] maximum incorrect');
AssertEquals_LREAL(0.046432387372313894, positionExtrema.Tmin, 1E-9, message:='Profile[2] Tmin incorrect');
AssertEquals_LREAL(58.396862666777764, positionExtrema.Minimum, 1E-9, message:='Profile[2] minimum incorrect');
   

TEST_FINISHED();
END_METHOD

METHOD Test_Trajectory_VelIntrf_HasMinDuration_HasTargetAcceleration_15
VAR_INST
  ruckig : Struckig.Otg(0.001, 3) := (
  
    ControlInterface := ControlInterfaceType.Velocity,
    Synchronization := SynchronizationType.TimeSync,
    MinDuration := 4.0,
    MaxVelocity := [ 2000.0, 2000.0, 2000.0 ],
    MaxAcceleration := [ 20000.0, 20000.0, 20000.0 ],
    MaxJerk := [ 800000.0, 800000.0, 800000.0 ],
    CurrentPosition := [ 75.56664126996091, 28.547892536688693, -86.85879483383854 ],
    CurrentVelocity := [ -907.5550785632845, -163.50892650730952, 945.093468981253 ],
    CurrentAcceleration := [ -9795.506987265866, -524.7660445364163, 6906.673195763407 ],
    TargetPosition := [ 55.76507784074343, -16.508527279558322, 66.12886627805486 ],
    TargetVelocity := [ 0.0, 0.0, 0.0 ],
    TargetAcceleration := [ 386.24278070399055, -278.2333273528002, 154.77366631011728 ]
  );
  
  positionExtrema : Struckig.ProfileBound;
END_VAR
TEST('Trajectory_VelIntrf_HasMinDuration_HasTargetAcceleration_15');

ruckig();

// Check total duration of profiles
AssertEquals_LREAL(Expected := 4.0, Actual := ruckig.Duration, DELTA := 1E-8, Message := 'Duration incorrect');

// Check minimum duration
AssertEquals_LREAL(Expected := ruckig.MinDuration, Actual := ruckig.Duration, DELTA := 1E-8, Message := 'Minimum duration not equals duration');

// Check duration for each phase
positionExtrema := ruckig._profiles[0].Bound();
AssertEquals_LREAL(0.0, positionExtrema.Tmax, 1E-9, message:='Profile[0] Tmax incorrect');
AssertEquals_LREAL(75.56664126996091, positionExtrema.Maximum, 1E-9, message:='Profile[0] maximum incorrect');
AssertEquals_LREAL(4.0, positionExtrema.Tmin, 1E-9, message:='Profile[0] Tmin incorrect');
AssertEquals_LREAL(-2987.772500918376, positionExtrema.Minimum, 1E-9, message:='Profile[0] minimum incorrect');

positionExtrema := ruckig._profiles[1].Bound();
AssertEquals_LREAL(0.0, positionExtrema.Tmax, 1E-9, message:='Profile[1] Tmax incorrect');
AssertEquals_LREAL(28.547892536688693, positionExtrema.Maximum, 1E-9, message:='Profile[1] maximum incorrect');
AssertEquals_LREAL(3.9996010293988298, positionExtrema.Tmin, 1E-9, message:='Profile[1] Tmin incorrect');
AssertEquals_LREAL(-298.7426270650857, positionExtrema.Minimum, 1E-9, message:='Profile[1] minimum incorrect');

positionExtrema := ruckig._profiles[2].Bound();
AssertEquals_LREAL(3.999613065832347, positionExtrema.Tmax, 1E-9, message:='Profile[2] Tmax incorrect');
AssertEquals_LREAL(1866.9541857476615, positionExtrema.Maximum, 1E-9, message:='Profile[2] maximum incorrect');
AssertEquals_LREAL(0.0, positionExtrema.Tmin, 1E-9, message:='Profile[2] Tmin incorrect');
AssertEquals_LREAL(-86.85879483383854, positionExtrema.Minimum, 1E-9, message:='Profile[2] minimum incorrect');
   

TEST_FINISHED();
END_METHOD

METHOD Test_Trajectory_VelIntrf_HasMinDuration_HasTargetAcceleration_2
VAR_INST
  ruckig : Struckig.Otg(0.001, 3) := (
  
    ControlInterface := ControlInterfaceType.Velocity,
    Synchronization := SynchronizationType.TimeSync,
    MinDuration := 9.0,
    MaxVelocity := [ 2000.0, 2000.0, 2000.0 ],
    MaxAcceleration := [ 20000.0, 20000.0, 20000.0 ],
    MaxJerk := [ 800000.0, 800000.0, 800000.0 ],
    CurrentPosition := [ -42.14366568546411, -0.17981567939382614, 52.710579417429415 ],
    CurrentVelocity := [ 907.7910933477099, -598.5253765205216, 843.5742135639091 ],
    CurrentAcceleration := [ -2130.463978487962, -4979.014587697566, 4505.077450884928 ],
    TargetPosition := [ -25.16463645590001, -87.36168316729645, -44.80074709880757 ],
    TargetVelocity := [ 0.0, 0.0, 0.0 ],
    TargetAcceleration := [ 135.9501252391201, 428.64680857177814, -269.3082926306902 ]
  );
  
  positionExtrema : Struckig.ProfileBound;
END_VAR
TEST('Trajectory_VelIntrf_HasMinDuration_HasTargetAcceleration_2');

ruckig();

// Check total duration of profiles
AssertEquals_LREAL(Expected := 9.0, Actual := ruckig.Duration, DELTA := 1E-8, Message := 'Duration incorrect');

// Check minimum duration
AssertEquals_LREAL(Expected := ruckig.MinDuration, Actual := ruckig.Duration, DELTA := 1E-8, Message := 'Minimum duration not equals duration');

// Check duration for each phase
positionExtrema := ruckig._profiles[0].Bound();
AssertEquals_LREAL(0.49554889236395766, positionExtrema.Tmax, 1E-9, message:='Profile[0] Tmax incorrect');
AssertEquals_LREAL(170.56370157598377, positionExtrema.Maximum, 1E-9, message:='Profile[0] maximum incorrect');
AssertEquals_LREAL(9.0, positionExtrema.Tmin, 1E-9, message:='Profile[0] Tmin incorrect');
AssertEquals_LREAL(-4211.910244370803, positionExtrema.Minimum, 1E-9, message:='Profile[0] minimum incorrect');

positionExtrema := ruckig._profiles[1].Bound();
AssertEquals_LREAL(0.0, positionExtrema.Tmax, 1E-9, message:='Profile[1] Tmax incorrect');
AssertEquals_LREAL(-0.17981567939382614, positionExtrema.Maximum, 1E-9, message:='Profile[1] maximum incorrect');
AssertEquals_LREAL(9.0, positionExtrema.Tmin, 1E-9, message:='Profile[1] Tmin incorrect');
AssertEquals_LREAL(-16050.750940855625, positionExtrema.Minimum, 1E-9, message:='Profile[1] minimum incorrect');

positionExtrema := ruckig._profiles[2].Bound();
AssertEquals_LREAL(9.0, positionExtrema.Tmax, 1E-9, message:='Profile[2] Tmax incorrect');
AssertEquals_LREAL(10611.025627794468, positionExtrema.Maximum, 1E-9, message:='Profile[2] maximum incorrect');
AssertEquals_LREAL(0.0, positionExtrema.Tmin, 1E-9, message:='Profile[2] Tmin incorrect');
AssertEquals_LREAL(52.710579417429415, positionExtrema.Minimum, 1E-9, message:='Profile[2] minimum incorrect');
   

TEST_FINISHED();
END_METHOD

METHOD Test_Trajectory_VelIntrf_HasMinDuration_HasTargetAcceleration_24
VAR_INST
  ruckig : Struckig.Otg(0.001, 3) := (
  
    ControlInterface := ControlInterfaceType.Velocity,
    Synchronization := SynchronizationType.TimeSync,
    MinDuration := 4.0,
    MaxVelocity := [ 2000.0, 2000.0, 2000.0 ],
    MaxAcceleration := [ 20000.0, 20000.0, 20000.0 ],
    MaxJerk := [ 800000.0, 800000.0, 800000.0 ],
    CurrentPosition := [ -36.09927130079986, -37.31605014687916, -21.87430633679142 ],
    CurrentVelocity := [ -860.5086573373251, 464.08652353185903, 200.18097757640635 ],
    CurrentAcceleration := [ -5460.19802538634, 6555.9925610093305, 3810.294831944326 ],
    TargetPosition := [ -54.24890759921874, -43.79874329759572, 97.31878234758045 ],
    TargetVelocity := [ 0.0, 0.0, 0.0 ],
    TargetAcceleration := [ 205.84209067138795, 982.2033443244447, 841.5190460798017 ]
  );
  
  positionExtrema : Struckig.ProfileBound;
END_VAR
TEST('Trajectory_VelIntrf_HasMinDuration_HasTargetAcceleration_24');

ruckig();

// Check total duration of profiles
AssertEquals_LREAL(Expected := 4.0, Actual := ruckig.Duration, DELTA := 1E-8, Message := 'Duration incorrect');

// Check minimum duration
AssertEquals_LREAL(Expected := ruckig.MinDuration, Actual := ruckig.Duration, DELTA := 1E-8, Message := 'Minimum duration not equals duration');

// Check duration for each phase
positionExtrema := ruckig._profiles[0].Bound();
AssertEquals_LREAL(0.0, positionExtrema.Tmax, 1E-9, message:='Profile[0] Tmax incorrect');
AssertEquals_LREAL(-36.09927130079986, positionExtrema.Maximum, 1E-9, message:='Profile[0] maximum incorrect');
AssertEquals_LREAL(3.9999999999994404, positionExtrema.Tmin, 1E-9, message:='Profile[0] Tmin incorrect');
AssertEquals_LREAL(-1797.4018084567545, positionExtrema.Minimum, 1E-9, message:='Profile[0] minimum incorrect');

positionExtrema := ruckig._profiles[1].Bound();
AssertEquals_LREAL(3.9986182669711527, positionExtrema.Tmax, 1E-9, message:='Profile[1] Tmax incorrect');
AssertEquals_LREAL(945.0172239763237, positionExtrema.Maximum, 1E-9, message:='Profile[1] maximum incorrect');
AssertEquals_LREAL(0.0, positionExtrema.Tmin, 1E-9, message:='Profile[1] Tmin incorrect');
AssertEquals_LREAL(-37.31605014687916, positionExtrema.Minimum, 1E-9, message:='Profile[1] minimum incorrect');

positionExtrema := ruckig._profiles[2].Bound();
AssertEquals_LREAL(3.998882474232829, positionExtrema.Tmax, 1E-9, message:='Profile[2] Tmax incorrect');
AssertEquals_LREAL(396.1255684695049, positionExtrema.Maximum, 1E-9, message:='Profile[2] maximum incorrect');
AssertEquals_LREAL(0.0, positionExtrema.Tmin, 1E-9, message:='Profile[2] Tmin incorrect');
AssertEquals_LREAL(-21.87430633679142, positionExtrema.Minimum, 1E-9, message:='Profile[2] minimum incorrect');
   

TEST_FINISHED();
END_METHOD

METHOD Test_Trajectory_VelIntrf_HasMinDuration_HasTargetAcceleration_28
VAR_INST
  ruckig : Struckig.Otg(0.001, 3) := (
  
    ControlInterface := ControlInterfaceType.Velocity,
    Synchronization := SynchronizationType.TimeSync,
    MinDuration := 1.0,
    MaxVelocity := [ 2000.0, 2000.0, 2000.0 ],
    MaxAcceleration := [ 20000.0, 20000.0, 20000.0 ],
    MaxJerk := [ 800000.0, 800000.0, 800000.0 ],
    CurrentPosition := [ 26.72988392867606, 89.87801257777275, -0.6552932842744923 ],
    CurrentVelocity := [ -910.1011363116729, 900.2984394511482, -861.6634451162208 ],
    CurrentAcceleration := [ -2119.6807052614504, 5529.302686481027, -4609.195103753672 ],
    TargetPosition := [ -39.13177680274664, 81.76531541204051, 73.56031276085977 ],
    TargetVelocity := [ 0.0, 0.0, 0.0 ],
    TargetAcceleration := [ -752.02419837743, -347.0115049647633, 917.7734303925099 ]
  );
  
  positionExtrema : Struckig.ProfileBound;
END_VAR
TEST('Trajectory_VelIntrf_HasMinDuration_HasTargetAcceleration_28');

ruckig();

// Check total duration of profiles
AssertEquals_LREAL(Expected := 1.0, Actual := ruckig.Duration, DELTA := 1E-8, Message := 'Duration incorrect');

// Check minimum duration
AssertEquals_LREAL(Expected := ruckig.MinDuration, Actual := ruckig.Duration, DELTA := 1E-8, Message := 'Minimum duration not equals duration');

// Check duration for each phase
positionExtrema := ruckig._profiles[0].Bound();
AssertEquals_LREAL(0.0, positionExtrema.Tmax, 1E-9, message:='Profile[0] Tmax incorrect');
AssertEquals_LREAL(26.72988392867606, positionExtrema.Maximum, 1E-9, message:='Profile[0] maximum incorrect');
AssertEquals_LREAL(0.9981199395040201, positionExtrema.Tmin, 1E-9, message:='Profile[0] Tmin incorrect');
AssertEquals_LREAL(-430.3267470254405, positionExtrema.Minimum, 1E-9, message:='Profile[0] minimum incorrect');

positionExtrema := ruckig._profiles[1].Bound();
AssertEquals_LREAL(1.0, positionExtrema.Tmax, 1E-9, message:='Profile[1] Tmax incorrect');
AssertEquals_LREAL(552.876667394997, positionExtrema.Maximum, 1E-9, message:='Profile[1] maximum incorrect');
AssertEquals_LREAL(0.0, positionExtrema.Tmin, 1E-9, message:='Profile[1] Tmin incorrect');
AssertEquals_LREAL(89.87801257777275, positionExtrema.Minimum, 1E-9, message:='Profile[1] minimum incorrect');

positionExtrema := ruckig._profiles[2].Bound();
AssertEquals_LREAL(0.0, positionExtrema.Tmax, 1E-9, message:='Profile[2] Tmax incorrect');
AssertEquals_LREAL(-0.6552932842744923, positionExtrema.Maximum, 1E-9, message:='Profile[2] maximum incorrect');
AssertEquals_LREAL(1.0, positionExtrema.Tmin, 1E-9, message:='Profile[2] Tmin incorrect');
AssertEquals_LREAL(-440.86209469106717, positionExtrema.Minimum, 1E-9, message:='Profile[2] minimum incorrect');
   

TEST_FINISHED();
END_METHOD

METHOD Test_Trajectory_VelIntrf_HasMinDuration_HasTargetVelocity_10
VAR_INST
  ruckig : Struckig.Otg(0.001, 3) := (
  
    ControlInterface := ControlInterfaceType.Velocity,
    Synchronization := SynchronizationType.TimeSync,
    MinDuration := 2.0,
    MaxVelocity := [ 2000.0, 2000.0, 2000.0 ],
    MaxAcceleration := [ 20000.0, 20000.0, 20000.0 ],
    MaxJerk := [ 800000.0, 800000.0, 800000.0 ],
    CurrentPosition := [ -51.10462658383166, 73.44882630640612, -19.30852635838795 ],
    CurrentVelocity := [ 164.50299939172464, -134.18423314468146, -464.3780778652133 ],
    CurrentAcceleration := [ -8278.692764283722, 6061.921891848055, 4386.12235664175 ],
    TargetPosition := [ 25.716005882813377, -70.06323197615777, -77.63731365300606 ],
    TargetVelocity := [ 860.5492611003563, -791.0913916516706, 153.1275749598924 ],
    TargetAcceleration := [ 0.0, 0.0, 0.0 ]
  );
  
  positionExtrema : Struckig.ProfileBound;
END_VAR
TEST('Trajectory_VelIntrf_HasMinDuration_HasTargetVelocity_10');

ruckig();

// Check total duration of profiles
AssertEquals_LREAL(Expected := 2.0, Actual := ruckig.Duration, DELTA := 1E-8, Message := 'Duration incorrect');

// Check minimum duration
AssertEquals_LREAL(Expected := ruckig.MinDuration, Actual := ruckig.Duration, DELTA := 1E-8, Message := 'Minimum duration not equals duration');

// Check duration for each phase
positionExtrema := ruckig._profiles[0].Bound();
AssertEquals_LREAL(2.0, positionExtrema.Tmax, 1E-9, message:='Profile[0] Tmax incorrect');
AssertEquals_LREAL(927.4368124889319, positionExtrema.Maximum, 1E-9, message:='Profile[0] maximum incorrect');
AssertEquals_LREAL(0.0, positionExtrema.Tmin, 1E-9, message:='Profile[0] Tmin incorrect');
AssertEquals_LREAL(-51.10462658383166, positionExtrema.Minimum, 1E-9, message:='Profile[0] minimum incorrect');

positionExtrema := ruckig._profiles[1].Bound();
AssertEquals_LREAL(0.0, positionExtrema.Tmax, 1E-9, message:='Profile[1] Tmax incorrect');
AssertEquals_LREAL(73.44882630640612, positionExtrema.Maximum, 1E-9, message:='Profile[1] maximum incorrect');
AssertEquals_LREAL(2.0, positionExtrema.Tmin, 1E-9, message:='Profile[1] Tmin incorrect');
AssertEquals_LREAL(-826.3421581283551, positionExtrema.Minimum, 1E-9, message:='Profile[1] minimum incorrect');

positionExtrema := ruckig._profiles[2].Bound();
AssertEquals_LREAL(2.0, positionExtrema.Tmax, 1E-9, message:='Profile[2] Tmax incorrect');
AssertEquals_LREAL(228.98909292790523, positionExtrema.Maximum, 1E-9, message:='Profile[2] maximum incorrect');
AssertEquals_LREAL(0.14135684112738017, positionExtrema.Tmin, 1E-9, message:='Profile[2] Tmin incorrect');
AssertEquals_LREAL(-48.46346696617425, positionExtrema.Minimum, 1E-9, message:='Profile[2] minimum incorrect');
   

TEST_FINISHED();
END_METHOD

METHOD Test_Trajectory_VelIntrf_HasMinDuration_HasTargetVelocity_29
VAR_INST
  ruckig : Struckig.Otg(0.001, 3) := (
  
    ControlInterface := ControlInterfaceType.Velocity,
    Synchronization := SynchronizationType.TimeSync,
    MinDuration := 2.0,
    MaxVelocity := [ 2000.0, 2000.0, 2000.0 ],
    MaxAcceleration := [ 20000.0, 20000.0, 20000.0 ],
    MaxJerk := [ 800000.0, 800000.0, 800000.0 ],
    CurrentPosition := [ -5.142966438749113, 46.38848214110482, 8.704597100063438 ],
    CurrentVelocity := [ 726.4037786608858, -283.30617235647094, 943.7013648213149 ],
    CurrentAcceleration := [ -9815.807193475257, 2003.8359857324049, 8221.03830030881 ],
    TargetPosition := [ 42.838039251838836, -59.62942353602521, -14.163596267977098 ],
    TargetVelocity := [ 780.2788462330652, -165.70194942906164, -320.9188038297459 ],
    TargetAcceleration := [ 0.0, 0.0, 0.0 ]
  );
  
  positionExtrema : Struckig.ProfileBound;
END_VAR
TEST('Trajectory_VelIntrf_HasMinDuration_HasTargetVelocity_29');

ruckig();

// Check total duration of profiles
AssertEquals_LREAL(Expected := 2.0, Actual := ruckig.Duration, DELTA := 1E-8, Message := 'Duration incorrect');

// Check minimum duration
AssertEquals_LREAL(Expected := ruckig.MinDuration, Actual := ruckig.Duration, DELTA := 1E-8, Message := 'Minimum duration not equals duration');

// Check duration for each phase
positionExtrema := ruckig._profiles[0].Bound();
AssertEquals_LREAL(2.0, positionExtrema.Tmax, 1E-9, message:='Profile[0] Tmax incorrect');
AssertEquals_LREAL(1440.8672021052723, positionExtrema.Maximum, 1E-9, message:='Profile[0] maximum incorrect');
AssertEquals_LREAL(0.0, positionExtrema.Tmin, 1E-9, message:='Profile[0] Tmin incorrect');
AssertEquals_LREAL(-5.142966438749113, positionExtrema.Minimum, 1E-9, message:='Profile[0] minimum incorrect');

positionExtrema := ruckig._profiles[1].Bound();
AssertEquals_LREAL(0.0, positionExtrema.Tmax, 1E-9, message:='Profile[1] Tmax incorrect');
AssertEquals_LREAL(46.38848214110482, positionExtrema.Maximum, 1E-9, message:='Profile[1] maximum incorrect');
AssertEquals_LREAL(2.0, positionExtrema.Tmin, 1E-9, message:='Profile[1] Tmin incorrect');
AssertEquals_LREAL(-289.6168422990306, positionExtrema.Minimum, 1E-9, message:='Profile[1] minimum incorrect');

positionExtrema := ruckig._profiles[2].Bound();
AssertEquals_LREAL(1.9991786543192867, positionExtrema.Tmax, 1E-9, message:='Profile[2] Tmax incorrect');
AssertEquals_LREAL(680.5617421837558, positionExtrema.Maximum, 1E-9, message:='Profile[2] maximum incorrect');
AssertEquals_LREAL(0.0, positionExtrema.Tmin, 1E-9, message:='Profile[2] Tmin incorrect');
AssertEquals_LREAL(8.704597100063438, positionExtrema.Minimum, 1E-9, message:='Profile[2] minimum incorrect');
   

TEST_FINISHED();
END_METHOD

METHOD Test_Trajectory_VelIntrf_HasMinDuration_HasTargetVelocity_31
VAR_INST
  ruckig : Struckig.Otg(0.001, 3) := (
  
    ControlInterface := ControlInterfaceType.Velocity,
    Synchronization := SynchronizationType.TimeSync,
    MinDuration := 1.0,
    MaxVelocity := [ 2000.0, 2000.0, 2000.0 ],
    MaxAcceleration := [ 20000.0, 20000.0, 20000.0 ],
    MaxJerk := [ 800000.0, 800000.0, 800000.0 ],
    CurrentPosition := [ 63.960578391499666, 54.48212252566097, -66.2665469971498 ],
    CurrentVelocity := [ -575.4579660082293, -11.705912611153622, -587.9381370421042 ],
    CurrentAcceleration := [ 8807.339705330302, 2358.7046624117775, 3594.3028645291306 ],
    TargetPosition := [ 22.667413933572206, 28.76217335632498, -66.10993276695004 ],
    TargetVelocity := [ 479.87839787357325, -385.01691049270346, 881.0646457402781 ],
    TargetAcceleration := [ 0.0, 0.0, 0.0 ]
  );
  
  positionExtrema : Struckig.ProfileBound;
END_VAR
TEST('Trajectory_VelIntrf_HasMinDuration_HasTargetVelocity_31');

ruckig();

// Check total duration of profiles
AssertEquals_LREAL(Expected := 1.0, Actual := ruckig.Duration, DELTA := 1E-8, Message := 'Duration incorrect');

// Check minimum duration
AssertEquals_LREAL(Expected := ruckig.MinDuration, Actual := ruckig.Duration, DELTA := 1E-8, Message := 'Minimum duration not equals duration');

// Check duration for each phase
positionExtrema := ruckig._profiles[0].Bound();
AssertEquals_LREAL(1.0, positionExtrema.Tmax, 1E-9, message:='Profile[0] Tmax incorrect');
AssertEquals_LREAL(459.53543867076246, positionExtrema.Maximum, 1E-9, message:='Profile[0] maximum incorrect');
AssertEquals_LREAL(0.07804745300795522, positionExtrema.Tmin, 1E-9, message:='Profile[0] Tmin incorrect');
AssertEquals_LREAL(42.96007142181631, positionExtrema.Minimum, 1E-9, message:='Profile[0] minimum incorrect');

positionExtrema := ruckig._profiles[1].Bound();
AssertEquals_LREAL(0.0, positionExtrema.Tmax, 1E-9, message:='Profile[1] Tmax incorrect');
AssertEquals_LREAL(54.48212252566097, positionExtrema.Maximum, 1E-9, message:='Profile[1] maximum incorrect');
AssertEquals_LREAL(1.0, positionExtrema.Tmin, 1E-9, message:='Profile[1] Tmin incorrect');
AssertEquals_LREAL(-141.58865895529902, positionExtrema.Minimum, 1E-9, message:='Profile[1] minimum incorrect');

positionExtrema := ruckig._profiles[2].Bound();
AssertEquals_LREAL(1.0, positionExtrema.Tmax, 1E-9, message:='Profile[2] Tmax incorrect');
AssertEquals_LREAL(414.54075498604016, positionExtrema.Maximum, 1E-9, message:='Profile[2] maximum incorrect');
AssertEquals_LREAL(0.1843671507002955, positionExtrema.Tmin, 1E-9, message:='Profile[2] Tmin incorrect');
AssertEquals_LREAL(-118.16839410819622, positionExtrema.Minimum, 1E-9, message:='Profile[2] minimum incorrect');
   

TEST_FINISHED();
END_METHOD

METHOD Test_Trajectory_VelIntrf_HasMinDuration_HasTargetVelocity_35
VAR_INST
  ruckig : Struckig.Otg(0.001, 3) := (
  
    ControlInterface := ControlInterfaceType.Velocity,
    Synchronization := SynchronizationType.TimeSync,
    MinDuration := 6.0,
    MaxVelocity := [ 2000.0, 2000.0, 2000.0 ],
    MaxAcceleration := [ 20000.0, 20000.0, 20000.0 ],
    MaxJerk := [ 800000.0, 800000.0, 800000.0 ],
    CurrentPosition := [ 86.79912594927566, -99.42921613569959, 73.84158750779326 ],
    CurrentVelocity := [ 452.6259236304402, -163.4023057855636, -304.0927897134642 ],
    CurrentAcceleration := [ -8056.463683684189, 1488.1788996032483, -5834.7185586681835 ],
    TargetPosition := [ -48.8659931716374, 95.30221236030337, -24.45741535022175 ],
    TargetVelocity := [ 764.7295518967278, 917.1744361726062, -421.38676355576445 ],
    TargetAcceleration := [ 0.0, 0.0, 0.0 ]
  );
  
  positionExtrema : Struckig.ProfileBound;
END_VAR
TEST('Trajectory_VelIntrf_HasMinDuration_HasTargetVelocity_35');

ruckig();

// Check total duration of profiles
AssertEquals_LREAL(Expected := 6.0, Actual := ruckig.Duration, DELTA := 1E-8, Message := 'Duration incorrect');

// Check minimum duration
AssertEquals_LREAL(Expected := ruckig.MinDuration, Actual := ruckig.Duration, DELTA := 1E-8, Message := 'Minimum duration not equals duration');

// Check duration for each phase
positionExtrema := ruckig._profiles[0].Bound();
AssertEquals_LREAL(6.0, positionExtrema.Tmax, 1E-9, message:='Profile[0] Tmax incorrect');
AssertEquals_LREAL(3615.5260437805628, positionExtrema.Maximum, 1E-9, message:='Profile[0] maximum incorrect');
AssertEquals_LREAL(0.0, positionExtrema.Tmin, 1E-9, message:='Profile[0] Tmin incorrect');
AssertEquals_LREAL(86.79912594927566, positionExtrema.Minimum, 1E-9, message:='Profile[0] minimum incorrect');

positionExtrema := ruckig._profiles[1].Bound();
AssertEquals_LREAL(6.0, positionExtrema.Tmax, 1E-9, message:='Profile[1] Tmax incorrect');
AssertEquals_LREAL(4880.54135783718, positionExtrema.Maximum, 1E-9, message:='Profile[1] maximum incorrect');
AssertEquals_LREAL(0.11429816171064022, positionExtrema.Tmin, 1E-9, message:='Profile[1] Tmin incorrect');
AssertEquals_LREAL(-108.6399927535293, positionExtrema.Minimum, 1E-9, message:='Profile[1] minimum incorrect');

